LIN {X 0.246,Y -561.732,Z 557.411,A 0.000,B 0.000,C 90.000,E1 109.939} C_DIS
LIN {X 0.060,Y -566.914,Z 557.408,A 0.000,B 0.000,C 90.000,E1 109.450} C_DIS
LIN {X 0.120,Y -571.794,Z 557.405,A 0.000,B 0.000,C 90.000,E1 108.906} C_DIS
LIN {X 0.026,Y -577.234,Z 557.401,A 0.000,B 0.000,C 90.000,E1 108.236} C_DIS
LIN {X 0.253,Y -582.926,Z 557.397,A 0.000,B 0.000,C 90.000,E1 107.402} C_DIS
LIN {X -0.014,Y -588.048,Z 557.392,A 0.000,B 0.000,C 90.000,E1 106.622} C_DIS
LIN {X 0.262,Y -593.519,Z 557.387,A 0.000,B 0.000,C 90.000,E1 105.662} C_DIS
LIN {X -0.063,Y -597.768,Z 557.383,A 0.000,B 0.000,C 90.000,E1 104.898} C_DIS
LIN {X 0.044,Y -603.619,Z 557.376,A 0.000,B 0.000,C 90.000,E1 103.703} C_DIS
LIN {X -0.051,Y -609.222,Z 557.370,A 0.000,B 0.000,C 90.000,E1 102.535} C_DIS
LIN {X -0.030,Y -612.189,Z 557.366,A 0.000,B 0.000,C 90.000,E1 101.883} C_DIS
LIN {X 0.063,Y -616.606,Z 557.360,A 0.000,B 0.000,C 90.000,E1 100.838} C_DIS
LIN {X -0.178,Y -617.680,Z 557.359,A 0.000,B 0.000,C 90.000,E1 100.602} C_DIS
LIN {X 0.226,Y -625.561,Z 557.347,A 0.000,B 0.000,C 90.000,E1 98.511} C_DIS
LIN {X 0.211,Y -630.523,Z 557.340,A 0.000,B 0.000,C 90.000,E1 97.239} C_DIS
LIN {X 0.129,Y -633.410,Z 557.336,A 0.000,B 0.000,C 90.000,E1 96.486} C_DIS
LIN {X -0.264,Y -636.936,Z 557.331,A 0.000,B 0.000,C 90.000,E1 95.511} C_DIS
LIN {X -0.295,Y -639.376,Z 557.326,A 0.000,B 0.000,C 90.000,E1 94.759} C_DIS
LIN {X 0.033,Y -642.183,Z 557.321,A 0.000,B 0.000,C 90.000,E1 93.726} C_DIS
LIN {X -0.005,Y -644.045,Z 557.317,A 0.000,B 0.000,C 90.000,E1 92.980} C_DIS
LIN {X -0.054,Y -645.623,Z 557.312,A 0.000,B 0.000,C 90.000,E1 92.236} C_DIS
LIN {X -0.063,Y -646.957,Z 557.308,A 0.000,B 0.000,C 90.000,E1 91.489} C_DIS
LIN {X 0.141,Y -647.672,Z 557.306,A 0.000,B 0.000,C 90.000,E1 90.974} C_DIS
LIN {X 0.136,Y -648.569,Z 557.301,A 0.000,B 0.000,C 90.000,E1 90.229} C_DIS
LIN {X -0.074,Y -649.177,Z 557.296,A 0.000,B 0.000,C 90.000,E1 89.255} C_DIS
LIN {X -0.289,Y -649.296,Z 557.294,A 0.000,B 0.000,C 90.000,E1 89.026} C_DIS
LIN {X 0.173,Y -649.169,Z 557.289,A 0.000,B 0.000,C 90.000,E1 87.993} C_DIS
LIN {X 0.177,Y -648.851,Z 557.285,A 0.000,B 0.000,C 90.000,E1 87.249} C_DIS
LIN {X -0.014,Y -647.981,Z 557.279,A 0.000,B 0.000,C 90.000,E1 86.274} C_DIS
LIN {X -0.218,Y -646.671,Z 557.274,A 0.000,B 0.000,C 90.000,E1 85.298} C_DIS
LIN {X 0.257,Y -645.100,Z 557.268,A 0.000,B 0.000,C 90.000,E1 84.261} C_DIS
LIN {X 0.246,Y -643.698,Z 557.264,A 0.000,B 0.000,C 90.000,E1 83.514} C_DIS
LIN {X 0.293,Y -641.950,Z 557.260,A 0.000,B 0.000,C 90.000,E1 82.761} C_DIS
LIN {X -0.109,Y -638.605,Z 557.253,A 0.000,B 0.000,C 90.000,E1 81.546} C_DIS
LIN {X -0.104,Y -636.298,Z 557.249,A 0.000,B 0.000,C 90.000,E1 80.792} C_DIS
LIN {X 0.317,Y -633.090,Z 557.243,A 0.000,B 0.000,C 90.000,E1 79.746} C_DIS
LIN {X 0.066,Y -629.496,Z 557.238,A 0.000,B 0.000,C 90.000,E1 78.757} C_DIS
LIN {X 0.095,Y -626.536,Z 557.233,A 0.000,B 0.000,C 90.000,E1 77.993} C_DIS
LIN {X -0.110,Y -622.314,Z 557.228,A 0.000,B 0.000,C 90.000,E1 76.992} C_DIS
LIN {X -0.147,Y -618.764,Z 557.223,A 0.000,B 0.000,C 90.000,E1 76.228} C_DIS
LIN {X 0.042,Y -616.906,Z 557.221,A 0.000,B 0.000,C 90.000,E1 75.825} C_DIS
LIN {X 0.133,Y -613.670,Z 557.218,A 0.000,B 0.000,C 90.000,E1 75.172} C_DIS
LIN {X -0.057,Y -608.690,Z 557.213,A 0.000,B 0.000,C 90.000,E1 74.283} C_DIS
LIN {X -0.085,Y -604.075,Z 557.208,A 0.000,B 0.000,C 90.000,E1 73.504} C_DIS
LIN {X 0.196,Y -600.066,Z 557.205,A 0.000,B 0.000,C 90.000,E1 72.851} C_DIS
LIN {X -0.124,Y -594.698,Z 557.201,A 0.000,B 0.000,C 90.000,E1 72.127} C_DIS
LIN {X -0.047,Y -589.323,Z 557.197,A 0.000,B 0.000,C 90.000,E1 71.456} C_DIS
LIN {X 0.057,Y -584.731,Z 557.194,A 0.000,B 0.000,C 90.000,E1 70.913} C_DIS
LIN {X 0.186,Y -579.750,Z 557.191,A 0.000,B 0.000,C 90.000,E1 70.369} C_DIS
LIN {X -0.324,Y -572.232,Z 557.187,A 0.000,B 0.000,C 90.000,E1 69.699} C_DIS
LIN {X -0.116,Y -568.454,Z 557.185,A 0.000,B 0.000,C 90.000,E1 69.337} C_DIS
LIN {X -0.234,Y -563.003,Z 557.183,A 0.000,B 0.000,C 90.000,E1 68.901} C_DIS
LIN {X -0.053,Y -558.351,Z 557.181,A 0.000,B 0.000,C 90.000,E1 68.539} C_DIS
LIN {X -0.168,Y -553.801,Z 557.179,A 0.000,B 0.000,C 90.000,E1 68.230} C_DIS
LIN {X -0.242,Y -547.427,Z 557.177,A 0.000,B 0.000,C 90.000,E1 67.847} C_DIS
LIN {X -0.026,Y -542.412,Z 557.175,A 0.000,B 0.000,C 90.000,E1 67.539} C_DIS
LIN {X -0.054,Y -537.211,Z 557.174,A 0.000,B 0.000,C 90.000,E1 67.283} C_DIS
LIN {X -0.161,Y -530.311,Z 557.172,A 0.000,B 0.000,C 90.000,E1 66.975} C_DIS
LIN {X 0.245,Y -519.773,Z 557.170,A 0.000,B 0.000,C 90.000,E1 66.485} C_DIS
LIN {X 0.121,Y -505.630,Z 557.167,A 0.000,B 0.000,C 90.000,E1 65.973} C_DIS
LIN {X 0.039,Y -487.939,Z 557.163,A 0.000,B 0.000,C 90.000,E1 65.357} C_DIS
LIN {X 0.281,Y -470.586,Z 557.160,A 0.000,B 0.000,C 90.000,E1 64.717} C_DIS
LIN {X -0.042,Y -459.761,Z 557.157,A 0.000,B 0.000,C 90.000,E1 64.332} C_DIS
LIN {X -0.076,Y -459.738,Z 557.157,A 0.000,B 0.000,C 90.000,E1 64.332} C_DIS
LIN {X -0.044,Y -455.591,Z 557.144,A 0.000,B 0.000,C 90.000,E1 61.975} C_DIS
LIN {X 0.139,Y -452.500,Z 557.137,A 0.000,B 0.000,C 90.000,E1 60.667} C_DIS
LIN {X -0.225,Y -443.899,Z 557.114,A 0.000,B 0.000,C 90.000,E1 56.501} C_DIS
LIN {X 0.022,Y -439.842,Z 557.105,A 0.000,B 0.000,C 90.000,E1 54.848} C_DIS
LIN {X -0.016,Y -439.846,Z 557.105,A 0.000,B 0.000,C 90.000,E1 54.848} C_DIS
LIN {X -0.142,Y -443.210,Z 557.092,A 0.000,B 0.000,C 90.000,E1 52.557} C_DIS
LIN {X 0.164,Y -445.597,Z 557.083,A 0.000,B 0.000,C 90.000,E1 50.884} C_DIS
LIN {X -0.172,Y -447.830,Z 557.074,A 0.000,B 0.000,C 90.000,E1 49.299} C_DIS
LIN {X 0.165,Y -450.382,Z 557.063,A 0.000,B 0.000,C 90.000,E1 47.310} C_DIS
LIN {X -0.114,Y -452.284,Z 557.054,A 0.000,B 0.000,C 90.000,E1 45.729} C_DIS
LIN {X -0.074,Y -453.265,Z 557.049,A 0.000,B 0.000,C 90.000,E1 44.757} C_DIS
LIN {X -0.025,Y -454.053,Z 557.043,A 0.000,B 0.000,C 90.000,E1 43.785} C_DIS
LIN {X -0.261,Y -454.800,Z 557.036,A 0.000,B 0.000,C 90.000,E1 42.528} C_DIS
LIN {X -0.149,Y -455.338,Z 557.029,A 0.000,B 0.000,C 90.000,E1 41.229} C_DIS
LIN {X -0.029,Y -455.588,Z 557.022,A 0.000,B 0.000,C 90.000,E1 39.930} C_DIS
LIN {X 0.152,Y -455.658,Z 557.015,A 0.000,B 0.000,C 90.000,E1 38.624} C_DIS
LIN {X -0.021,Y -455.585,Z 557.008,A 0.000,B 0.000,C 90.000,E1 37.363} C_DIS
LIN {X 0.249,Y -455.272,Z 556.999,A 0.000,B 0.000,C 90.000,E1 35.724} C_DIS
LIN {X 0.246,Y -454.649,Z 556.990,A 0.000,B 0.000,C 90.000,E1 34.119} C_DIS
LIN {X -0.020,Y -454.134,Z 556.981,A 0.000,B 0.000,C 90.000,E1 32.546} C_DIS
LIN {X 0.183,Y -453.549,Z 556.970,A 0.000,B 0.000,C 90.000,E1 30.590} C_DIS
LIN {X 0.040,Y -453.118,Z 556.961,A 0.000,B 0.000,C 90.000,E1 28.999} C_DIS
LIN {X 0.068,Y -452.621,Z 556.952,A 0.000,B 0.000,C 90.000,E1 27.385} C_DIS
LIN {X 0.121,Y -452.373,Z 556.947,A 0.000,B 0.000,C 90.000,E1 26.411} C_DIS
LIN {X 0.115,Y -451.771,Z 556.934,A 0.000,B 0.000,C 90.000,E1 24.155} C_DIS
LIN {X 0.211,Y -451.371,Z 556.924,A 0.000,B 0.000,C 90.000,E1 22.206} C_DIS
LIN {X -0.167,Y -451.125,Z 556.911,A 0.000,B 0.000,C 90.000,E1 19.993} C_DIS
LIN {X 0.141,Y -451.053,Z 556.898,A 0.000,B 0.000,C 90.000,E1 17.692} C_DIS
LIN {X 0.179,Y -451.171,Z 556.886,A 0.000,B 0.000,C 90.000,E1 15.426} C_DIS
LIN {X 0.056,Y -451.742,Z 556.870,A 0.000,B 0.000,C 90.000,E1 12.535} C_DIS
LIN {X -0.002,Y -452.722,Z 556.855,A 0.000,B 0.000,C 90.000,E1 9.962} C_DIS
LIN {X 0.047,Y -453.845,Z 556.843,A 0.000,B 0.000,C 90.000,E1 7.701} C_DIS
LIN {X -0.149,Y -455.117,Z 556.832,A 0.000,B 0.000,C 90.000,E1 5.796} C_DIS
LIN {X -0.007,Y -456.994,Z 556.818,A 0.000,B 0.000,C 90.000,E1 3.212} C_DIS
LIN {X -0.085,Y -460.624,Z 556.797,A 0.000,B 0.000,C 90.000,E1 359.484} C_DIS
LIN {X 0.195,Y -463.699,Z 556.783,A 0.000,B 0.000,C 90.000,E1 356.906} C_DIS
LIN {X 0.192,Y -467.221,Z 556.769,A 0.000,B 0.000,C 90.000,E1 354.375} C_DIS
LIN {X -0.148,Y -469.847,Z 556.758,A 0.000,B 0.000,C 90.000,E1 352.527} C_DIS
LIN {X 0.030,Y -472.470,Z 556.748,A 0.000,B 0.000,C 90.000,E1 350.622} C_DIS
LIN {X 0.086,Y -476.234,Z 556.734,A 0.000,B 0.000,C 90.000,E1 348.117} C_DIS
LIN {X -0.171,Y -479.221,Z 556.724,A 0.000,B 0.000,C 90.000,E1 346.284} C_DIS
LIN {X 0.115,Y -482.419,Z 556.713,A 0.000,B 0.000,C 90.000,E1 344.393} C_DIS
LIN {X 0.000,Y -487.004,Z 556.700,A 0.000,B 0.000,C 90.000,E1 341.945} C_DIS
LIN {X -0.067,Y -490.007,Z 556.691,A 0.000,B 0.000,C 90.000,E1 340.423} C_DIS
LIN {X -0.073,Y -492.971,Z 556.683,A 0.000,B 0.000,C 90.000,E1 338.901} C_DIS
LIN {X 0.150,Y -495.863,Z 556.674,A 0.000,B 0.000,C 90.000,E1 337.358} C_DIS
LIN {X -0.036,Y -498.677,Z 556.666,A 0.000,B 0.000,C 90.000,E1 335.869} C_DIS
LIN {X 0.028,Y -501.386,Z 556.658,A 0.000,B 0.000,C 90.000,E1 334.357} C_DIS
LIN {X -0.087,Y -503.959,Z 556.649,A 0.000,B 0.000,C 90.000,E1 332.871} C_DIS
LIN {X -0.151,Y -506.459,Z 556.641,A 0.000,B 0.000,C 90.000,E1 331.385} C_DIS
LIN {X -0.037,Y -509.523,Z 556.631,A 0.000,B 0.000,C 90.000,E1 329.587} C_DIS
LIN {X 0.152,Y -512.579,Z 556.621,A 0.000,B 0.000,C 90.000,E1 327.788} C_DIS
LIN {X -0.109,Y -515.163,Z 556.613,A 0.000,B 0.000,C 90.000,E1 326.342} C_DIS
LIN {X 0.099,Y -517.782,Z 556.605,A 0.000,B 0.000,C 90.000,E1 324.848} C_DIS
LIN {X -0.253,Y -520.828,Z 556.595,A 0.000,B 0.000,C 90.000,E1 323.130} C_DIS
LIN {X -0.296,Y -525.163,Z 556.582,A 0.000,B 0.000,C 90.000,E1 320.803} C_DIS
LIN {X -0.057,Y -531.883,Z 556.564,A 0.000,B 0.000,C 90.000,E1 317.595} C_DIS
LIN {X -0.283,Y -537.412,Z 556.552,A 0.000,B 0.000,C 90.000,E1 315.324} C_DIS
LIN {X 0.025,Y -540.889,Z 556.544,A 0.000,B 0.000,C 90.000,E1 313.866} C_DIS
LIN {X 0.042,Y -545.394,Z 556.534,A 0.000,B 0.000,C 90.000,E1 312.162} C_DIS
LIN {X 0.055,Y -547.077,Z 556.531,A 0.000,B 0.000,C 90.000,E1 311.595} C_DIS
LIN {X 0.090,Y -547.862,Z 556.530,A 0.000,B 0.000,C 90.000,E1 311.310} C_DIS
LIN {X -0.250,Y -548.890,Z 556.528,A 0.000,B 0.000,C 90.000,E1 311.067} C_DIS
LIN {X -0.208,Y -549.690,Z 556.526,A 0.000,B 0.000,C 90.000,E1 310.782} C_DIS
LIN {X -0.006,Y -550.225,Z 556.526,A 0.000,B 0.000,C 90.000,E1 310.620} C_DIS
LIN {X 0.248,Y -552.243,Z 556.523,A 0.000,B 0.000,C 90.000,E1 310.172} C_DIS
LIN {X -0.031,Y -554.556,Z 556.521,A 0.000,B 0.000,C 90.000,E1 309.850} C_DIS
LIN {X -0.106,Y -557.886,Z 556.519,A 0.000,B 0.000,C 90.000,E1 309.439} C_DIS
LIN {X 0.084,Y -562.492,Z 556.517,A 0.000,B 0.000,C 90.000,E1 308.955} C_DIS
LIN {X 0.103,Y -570.439,Z 556.513,A 0.000,B 0.000,C 90.000,E1 308.302} C_DIS
LIN {X 0.290,Y -580.640,Z 556.509,A 0.000,B 0.000,C 90.000,E1 307.523} C_DIS
LIN {X -0.049,Y -587.620,Z 556.506,A 0.000,B 0.000,C 90.000,E1 306.996} C_DIS
LIN {X -0.167,Y -591.705,Z 556.504,A 0.000,B 0.000,C 90.000,E1 306.664} C_DIS
LIN {X -0.083,Y -596.826,Z 556.501,A 0.000,B 0.000,C 90.000,E1 306.171} C_DIS
LIN {X 0.120,Y -601.796,Z 556.498,A 0.000,B 0.000,C 90.000,E1 305.644} C_DIS
LIN {X -0.162,Y -609.169,Z 556.494,A 0.000,B 0.000,C 90.000,E1 304.898} C_DIS
LIN {X -0.120,Y -615.082,Z 556.490,A 0.000,B 0.000,C 90.000,E1 304.246} C_DIS
LIN {X 0.101,Y -622.014,Z 556.486,A 0.000,B 0.000,C 90.000,E1 303.452} C_DIS
LIN {X -0.118,Y -627.486,Z 556.482,A 0.000,B 0.000,C 90.000,E1 302.832} C_DIS
LIN {X -0.294,Y -632.694,Z 556.479,A 0.000,B 0.000,C 90.000,E1 302.212} C_DIS
LIN {X 0.108,Y -637.456,Z 556.475,A 0.000,B 0.000,C 90.000,E1 301.544} C_DIS
LIN {X 0.008,Y -641.457,Z 556.472,A 0.000,B 0.000,C 90.000,E1 300.924} C_DIS
LIN {X 0.129,Y -644.378,Z 556.469,A 0.000,B 0.000,C 90.000,E1 300.413} C_DIS
LIN {X 0.075,Y -647.411,Z 556.466,A 0.000,B 0.000,C 90.000,E1 299.795} C_DIS
LIN {X -0.238,Y -650.507,Z 556.461,A 0.000,B 0.000,C 90.000,E1 299.077} C_DIS
LIN {X 0.053,Y -653.212,Z 556.457,A 0.000,B 0.000,C 90.000,E1 298.309} C_DIS
LIN {X -0.089,Y -656.682,Z 556.452,A 0.000,B 0.000,C 90.000,E1 297.334} C_DIS
LIN {X 0.029,Y -657.730,Z 556.451,A 0.000,B 0.000,C 90.000,E1 297.078} C_DIS
LIN {X 0.151,Y -658.625,Z 556.449,A 0.000,B 0.000,C 90.000,E1 296.821} C_DIS
LIN {X -0.189,Y -660.124,Z 556.446,A 0.000,B 0.000,C 90.000,E1 296.360} C_DIS
LIN {X -0.059,Y -660.614,Z 556.445,A 0.000,B 0.000,C 90.000,E1 296.104} C_DIS
LIN {X 0.205,Y -660.847,Z 556.442,A 0.000,B 0.000,C 90.000,E1 295.591} C_DIS
LIN {X 0.336,Y -660.497,Z 556.441,A 0.000,B 0.000,C 90.000,E1 295.335} C_DIS
LIN {X 0.402,Y -659.757,Z 556.440,A 0.000,B 0.000,C 90.000,E1 295.207} C_DIS
LIN {X -0.409,Y -659.189,Z 556.440,A 0.000,B 0.000,C 90.000,E1 295.155} C_DIS
LIN {X 0.085,Y -658.729,Z 556.439,A 0.000,B 0.000,C 90.000,E1 294.975} C_DIS
LIN {X 0.213,Y -657.506,Z 556.438,A 0.000,B 0.000,C 90.000,E1 294.719} C_DIS
LIN {X -0.130,Y -653.750,Z 556.435,A 0.000,B 0.000,C 90.000,E1 294.387} C_DIS
LIN {X -0.002,Y -652.702,Z 556.435,A 0.000,B 0.000,C 90.000,E1 294.259} C_DIS
LIN {X 0.050,Y -651.126,Z 556.434,A 0.000,B 0.000,C 90.000,E1 294.131} C_DIS
LIN {X -0.092,Y -644.023,Z 556.432,A 0.000,B 0.000,C 90.000,E1 293.770} C_DIS
LIN {X -0.176,Y -642.024,Z 556.432,A 0.000,B 0.000,C 90.000,E1 293.695} C_DIS
LIN {X -0.331,Y -636.032,Z 556.431,A 0.000,B 0.000,C 90.000,E1 293.515} C_DIS
LIN {X 0.086,Y -632.311,Z 556.430,A 0.000,B 0.000,C 90.000,E1 293.334} C_DIS
LIN {X -0.236,Y -621.253,Z 556.428,A 0.000,B 0.000,C 90.000,E1 293.025} C_DIS
LIN {X 0.165,Y -617.083,Z 556.427,A 0.000,B 0.000,C 90.000,E1 292.845} C_DIS
LIN {X -0.060,Y -587.800,Z 556.422,A 0.000,B 0.000,C 90.000,E1 291.950} C_DIS
LIN {X -0.084,Y -579.731,Z 556.420,A 0.000,B 0.000,C 90.000,E1 291.663} C_DIS
LIN {X -0.040,Y -574.163,Z 556.419,A 0.000,B 0.000,C 90.000,E1 291.408} C_DIS
LIN {X -0.185,Y -569.857,Z 556.417,A 0.000,B 0.000,C 90.000,E1 291.153} C_DIS
LIN {X 0.029,Y -568.280,Z 556.416,A 0.000,B 0.000,C 90.000,E1 290.918} C_DIS
LIN {X 0.013,Y -567.693,Z 556.415,A 0.000,B 0.000,C 90.000,E1 290.663} C_DIS
LIN {X -0.039,Y -567.413,Z 556.412,A 0.000,B 0.000,C 90.000,E1 290.120} C_DIS
LIN {X 0.198,Y -567.328,Z 556.404,A 0.000,B 0.000,C 90.000,E1 288.725} C_DIS
LIN {X 0.097,Y -567.175,Z 556.398,A 0.000,B 0.000,C 90.000,E1 287.638} C_DIS
LIN {X 0.151,Y -566.751,Z 556.390,A 0.000,B 0.000,C 90.000,E1 286.260} C_DIS
LIN {X -0.193,Y -565.873,Z 556.381,A 0.000,B 0.000,C 90.000,E1 284.647} C_DIS
LIN {X 0.094,Y -565.058,Z 556.374,A 0.000,B 0.000,C 90.000,E1 283.244} C_DIS
LIN {X -0.053,Y -564.308,Z 556.366,A 0.000,B 0.000,C 90.000,E1 281.883} C_DIS
LIN {X 0.106,Y -563.565,Z 556.358,A 0.000,B 0.000,C 90.000,E1 280.489} C_DIS
LIN {X 0.020,Y -562.571,Z 556.348,A 0.000,B 0.000,C 90.000,E1 278.568} C_DIS
LIN {X -0.256,Y -561.703,Z 556.337,A 0.000,B 0.000,C 90.000,E1 276.663} C_DIS
LIN {X 0.114,Y -561.352,Z 556.332,A 0.000,B 0.000,C 90.000,E1 275.796} C_DIS
LIN {X 0.088,Y -560.796,Z 556.325,A 0.000,B 0.000,C 90.000,E1 274.416} C_DIS
LIN {X 0.047,Y -560.239,Z 556.317,A 0.000,B 0.000,C 90.000,E1 273.037} C_DIS
LIN {X 0.142,Y -559.423,Z 556.306,A 0.000,B 0.000,C 90.000,E1 271.088} C_DIS
LIN {X 0.034,Y -558.715,Z 556.298,A 0.000,B 0.000,C 90.000,E1 269.714} C_DIS
LIN {X 0.096,Y -557.677,Z 556.288,A 0.000,B 0.000,C 90.000,E1 267.764} C_DIS
LIN {X -0.029,Y -556.879,Z 556.280,A 0.000,B 0.000,C 90.000,E1 266.388} C_DIS
LIN {X -0.066,Y -555.872,Z 556.271,A 0.000,B 0.000,C 90.000,E1 264.723} C_DIS
LIN {X -0.079,Y -554.755,Z 556.261,A 0.000,B 0.000,C 90.000,E1 263.053} C_DIS
LIN {X -0.092,Y -553.759,Z 556.254,A 0.000,B 0.000,C 90.000,E1 261.659} C_DIS
LIN {X -0.204,Y -552.293,Z 556.246,A 0.000,B 0.000,C 90.000,E1 260.274} C_DIS
LIN {X 0.180,Y -549.638,Z 556.233,A 0.000,B 0.000,C 90.000,E1 257.993} C_DIS
LIN {X -0.252,Y -547.788,Z 556.224,A 0.000,B 0.000,C 90.000,E1 256.353} C_DIS
LIN {X 0.068,Y -545.677,Z 556.215,A 0.000,B 0.000,C 90.000,E1 254.629} C_DIS
LIN {X -0.049,Y -544.507,Z 556.210,A 0.000,B 0.000,C 90.000,E1 253.795} C_DIS
LIN {X -0.327,Y -541.934,Z 556.201,A 0.000,B 0.000,C 90.000,E1 252.127} C_DIS
LIN {X -0.094,Y -540.044,Z 556.194,A 0.000,B 0.000,C 90.000,E1 250.967} C_DIS
LIN {X -0.066,Y -538.087,Z 556.188,A 0.000,B 0.000,C 90.000,E1 249.826} C_DIS
LIN {X -0.178,Y -535.280,Z 556.180,A 0.000,B 0.000,C 90.000,E1 248.411} C_DIS
LIN {X 0.154,Y -532.886,Z 556.174,A 0.000,B 0.000,C 90.000,E1 247.230} C_DIS
LIN {X -0.035,Y -530.386,Z 556.167,A 0.000,B 0.000,C 90.000,E1 246.102} C_DIS
LIN {X -0.259,Y -527.720,Z 556.161,A 0.000,B 0.000,C 90.000,E1 244.973} C_DIS
LIN {X -0.133,Y -524.130,Z 556.153,A 0.000,B 0.000,C 90.000,E1 243.512} C_DIS
LIN {X 0.159,Y -520.389,Z 556.145,A 0.000,B 0.000,C 90.000,E1 242.025} C_DIS
LIN {X -0.077,Y -516.643,Z 556.137,A 0.000,B 0.000,C 90.000,E1 240.589} C_DIS
LIN {X -0.037,Y -513.407,Z 556.130,A 0.000,B 0.000,C 90.000,E1 239.410} C_DIS
LIN {X -0.252,Y -507.950,Z 556.120,A 0.000,B 0.000,C 90.000,E1 237.661} C_DIS
LIN {X -0.127,Y -501.004,Z 556.107,A 0.000,B 0.000,C 90.000,E1 235.261} C_DIS
LIN {X -0.187,Y -493.404,Z 556.092,A 0.000,B 0.000,C 90.000,E1 232.557} C_DIS
LIN {X 0.064,Y -489.298,Z 556.083,A 0.000,B 0.000,C 90.000,E1 231.009} C_DIS
LIN {X 0.236,Y -485.378,Z 556.075,A 0.000,B 0.000,C 90.000,E1 229.461} C_DIS
LIN {X 0.081,Y -480.635,Z 556.065,A 0.000,B 0.000,C 90.000,E1 227.634} C_DIS
LIN {X 0.013,Y -474.464,Z 556.051,A 0.000,B 0.000,C 90.000,E1 225.162} C_DIS
LIN {X -0.167,Y -470.788,Z 556.042,A 0.000,B 0.000,C 90.000,E1 223.623} C_DIS
LIN {X 0.091,Y -465.675,Z 556.030,A 0.000,B 0.000,C 90.000,E1 221.391} C_DIS
LIN {X -0.093,Y -460.693,Z 556.018,A 0.000,B 0.000,C 90.000,E1 219.197} C_DIS
LIN {X -0.083,Y -456.527,Z 556.007,A 0.000,B 0.000,C 90.000,E1 217.282} C_DIS
LIN {X 0.082,Y -451.106,Z 555.993,A 0.000,B 0.000,C 90.000,E1 214.692} C_DIS
LIN {X 0.137,Y -446.542,Z 555.980,A 0.000,B 0.000,C 90.000,E1 212.418} C_DIS
LIN {X 0.251,Y -441.609,Z 555.966,A 0.000,B 0.000,C 90.000,E1 209.795} C_DIS
LIN {X -0.056,Y -436.924,Z 555.951,A 0.000,B 0.000,C 90.000,E1 207.206} C_DIS
LIN {X 0.224,Y -434.723,Z 555.944,A 0.000,B 0.000,C 90.000,E1 205.848} C_DIS
LIN {X 0.092,Y -431.993,Z 555.935,A 0.000,B 0.000,C 90.000,E1 204.207} C_DIS
LIN {X -0.086,Y -428.371,Z 555.922,A 0.000,B 0.000,C 90.000,E1 201.897} C_DIS
LIN {X -0.083,Y -424.536,Z 555.907,A 0.000,B 0.000,C 90.000,E1 199.214} C_DIS
LIN {X 0.052,Y -422.347,Z 555.897,A 0.000,B 0.000,C 90.000,E1 197.511} C_DIS
LIN {X 0.055,Y -419.752,Z 555.886,A 0.000,B 0.000,C 90.000,E1 195.481} C_DIS
LIN {X 0.138,Y -417.820,Z 555.877,A 0.000,B 0.000,C 90.000,E1 193.772} C_DIS
LIN {X -0.009,Y -416.441,Z 555.871,A 0.000,B 0.000,C 90.000,E1 192.771} C_DIS
LIN {X -0.165,Y -411.538,Z 555.850,A 0.000,B 0.000,C 90.000,E1 189.029} C_DIS
LIN {X -0.031,Y -408.211,Z 555.833,A 0.000,B 0.000,C 90.000,E1 185.910} C_DIS
LIN {X -0.056,Y -406.914,Z 555.825,A 0.000,B 0.000,C 90.000,E1 184.531} C_DIS
LIN {X 0.142,Y -403.757,Z 555.806,A 0.000,B 0.000,C 90.000,E1 181.031} C_DIS
LIN {X -0.160,Y -401.745,Z 555.788,A 0.000,B 0.000,C 90.000,E1 177.936} C_DIS
LIN {X -0.043,Y -400.547,Z 555.773,A 0.000,B 0.000,C 90.000,E1 175.122} C_DIS
LIN {X 0.088,Y -399.857,Z 555.755,A 0.000,B 0.000,C 90.000,E1 171.951} C_DIS
LIN {X 0.009,Y -399.774,Z 555.744,A 0.000,B 0.000,C 90.000,E1 169.859} C_DIS
LIN {X -0.035,Y -399.964,Z 555.728,A 0.000,B 0.000,C 90.000,E1 167.061} C_DIS
LIN {X 0.127,Y -400.385,Z 555.716,A 0.000,B 0.000,C 90.000,E1 164.936} C_DIS
LIN {X -0.193,Y -401.346,Z 555.701,A 0.000,B 0.000,C 90.000,E1 162.181} C_DIS
LIN {X 0.059,Y -402.428,Z 555.687,A 0.000,B 0.000,C 90.000,E1 159.699} C_DIS
LIN {X -0.124,Y -403.678,Z 555.674,A 0.000,B 0.000,C 90.000,E1 157.283} C_DIS
LIN {X -0.111,Y -405.118,Z 555.660,A 0.000,B 0.000,C 90.000,E1 154.845} C_DIS
LIN {X 0.014,Y -406.362,Z 555.649,A 0.000,B 0.000,C 90.000,E1 152.743} C_DIS
LIN {X 0.077,Y -407.396,Z 555.639,A 0.000,B 0.000,C 90.000,E1 151.001} C_DIS
LIN {X -0.003,Y -408.278,Z 555.629,A 0.000,B 0.000,C 90.000,E1 149.282} C_DIS
LIN {X -0.119,Y -408.845,Z 555.622,A 0.000,B 0.000,C 90.000,E1 147.916} C_DIS
LIN {X 0.122,Y -409.336,Z 555.614,A 0.000,B 0.000,C 90.000,E1 146.501} C_DIS
LIN {X 0.021,Y -409.833,Z 555.606,A 0.000,B 0.000,C 90.000,E1 145.135} C_DIS
LIN {X 0.137,Y -410.260,Z 555.595,A 0.000,B 0.000,C 90.000,E1 143.050} C_DIS
LIN {X 0.108,Y -410.492,Z 555.585,A 0.000,B 0.000,C 90.000,E1 141.331} C_DIS
LIN {X 0.013,Y -410.605,Z 555.576,A 0.000,B 0.000,C 90.000,E1 139.622} C_DIS
LIN {X 0.037,Y -410.644,Z 555.564,A 0.000,B 0.000,C 90.000,E1 137.553} C_DIS
LIN {X 0.042,Y -410.739,Z 555.553,A 0.000,B 0.000,C 90.000,E1 135.486} C_DIS
LIN {X -0.099,Y -410.948,Z 555.543,A 0.000,B 0.000,C 90.000,E1 133.785} C_DIS
LIN {X 0.054,Y -411.122,Z 555.534,A 0.000,B 0.000,C 90.000,E1 132.043} C_DIS
LIN {X -0.194,Y -411.095,Z 555.526,A 0.000,B 0.000,C 90.000,E1 130.701} C_DIS
LIN {X 0.143,Y -410.907,Z 555.518,A 0.000,B 0.000,C 90.000,E1 129.277} C_DIS
LIN {X 0.055,Y -410.617,Z 555.513,A 0.000,B 0.000,C 90.000,E1 128.257} C_DIS
LIN {X -0.211,Y -410.410,Z 555.510,A 0.000,B 0.000,C 90.000,E1 127.729} C_DIS
LIN {X 0.075,Y -410.416,Z 555.509,A 0.000,B 0.000,C 90.000,E1 127.684} C_DIS
LIN {X -0.190,Y -415.820,Z 555.499,A 0.000,B 0.000,C 90.000,E1 125.884} C_DIS
LIN {X -0.086,Y -425.279,Z 555.479,A 0.000,B 0.000,C 90.000,E1 122.133} C_DIS
LIN {X -0.152,Y -430.286,Z 555.469,A 0.000,B 0.000,C 90.000,E1 120.463} C_DIS
LIN {X -0.154,Y -431.177,Z 555.467,A 0.000,B 0.000,C 90.000,E1 120.129} C_DIS
LIN {X -0.135,Y -440.845,Z 555.446,A 0.000,B 0.000,C 90.000,E1 116.283} C_DIS
LIN {X 0.221,Y -440.859,Z 555.446,A 0.000,B 0.000,C 90.000,E1 116.232} C_DIS
LIN {X 0.181,Y -440.903,Z 555.446,A 0.000,B 0.000,C 90.000,E1 116.232} C_DIS
LIN {X -0.201,Y -466.035,Z 555.440,A 0.000,B 0.000,C 90.000,E1 115.155} C_DIS
LIN {X -0.089,Y -481.629,Z 555.436,A 0.000,B 0.000,C 90.000,E1 114.463} C_DIS
LIN {X 0.121,Y -495.089,Z 555.432,A 0.000,B 0.000,C 90.000,E1 113.823} C_DIS
LIN {X 0.140,Y -505.135,Z 555.430,A 0.000,B 0.000,C 90.000,E1 113.334} C_DIS
LIN {X -0.211,Y -516.700,Z 555.426,A 0.000,B 0.000,C 90.000,E1 112.770} C_DIS
LIN {X 0.174,Y -521.670,Z 555.425,A 0.000,B 0.000,C 90.000,E1 112.461} C_DIS
LIN {X -0.010,Y -532.926,Z 555.421,A 0.000,B 0.000,C 90.000,E1 111.844} C_DIS
LIN {X 0.006,Y -539.270,Z 555.419,A 0.000,B 0.000,C 90.000,E1 111.461} C_DIS
LIN {X 0.146,Y -545.378,Z 555.417,A 0.000,B 0.000,C 90.000,E1 111.046} C_DIS
LIN {X 0.291,Y -551.315,Z 555.415,A 0.000,B 0.000,C 90.000,E1 110.610} C_DIS
LIN {X 0.091,Y -555.703,Z 555.413,A 0.000,B 0.000,C 90.000,E1 110.301} C_DIS
LIN {X -0.189,Y -561.189,Z 555.410,A 0.000,B 0.000,C 90.000,E1 109.866} C_DIS
LIN {X 0.259,Y -566.391,Z 555.408,A 0.000,B 0.000,C 90.000,E1 109.322} C_DIS
LIN {X -0.078,Y -571.276,Z 555.405,A 0.000,B 0.000,C 90.000,E1 108.833} C_DIS
LIN {X 0.330,Y -577.300,Z 555.401,A 0.000,B 0.000,C 90.000,E1 108.055} C_DIS
LIN {X -0.118,Y -580.266,Z 555.398,A 0.000,B 0.000,C 90.000,E1 107.692} C_DIS
LIN {X 0.087,Y -582.263,Z 555.397,A 0.000,B 0.000,C 90.000,E1 107.402} C_DIS
LIN {X -0.268,Y -588.417,Z 555.392,A 0.000,B 0.000,C 90.000,E1 106.496} C_DIS
LIN {X -0.153,Y -594.014,Z 555.386,A 0.000,B 0.000,C 90.000,E1 105.552} C_DIS
LIN {X 0.191,Y -598.977,Z 555.381,A 0.000,B 0.000,C 90.000,E1 104.592} C_DIS
LIN {X -0.145,Y -603.623,Z 555.376,A 0.000,B 0.000,C 90.000,E1 103.703} C_DIS
LIN {X -0.240,Y -609.386,Z 555.370,A 0.000,B 0.000,C 90.000,E1 102.535} C_DIS
LIN {X 0.195,Y -612.997,Z 555.365,A 0.000,B 0.000,C 90.000,E1 101.715} C_DIS
LIN {X 0.057,Y -616.393,Z 555.361,A 0.000,B 0.000,C 90.000,E1 100.950} C_DIS
LIN {X 0.071,Y -618.507,Z 555.358,A 0.000,B 0.000,C 90.000,E1 100.433} C_DIS
LIN {X 0.295,Y -627.505,Z 555.345,A 0.000,B 0.000,C 90.000,E1 98.106} C_DIS
LIN {X 0.313,Y -632.469,Z 555.338,A 0.000,B 0.000,C 90.000,E1 96.834} C_DIS
LIN {X -0.025,Y -636.225,Z 555.333,A 0.000,B 0.000,C 90.000,E1 95.853} C_DIS
LIN {X 0.261,Y -639.538,Z 555.327,A 0.000,B 0.000,C 90.000,E1 94.821} C_DIS
LIN {X -0.189,Y -641.071,Z 555.324,A 0.000,B 0.000,C 90.000,E1 94.359} C_DIS
LIN {X -0.234,Y -643.150,Z 555.320,A 0.000,B 0.000,C 90.000,E1 93.612} C_DIS
LIN {X -0.263,Y -644.999,Z 555.316,A 0.000,B 0.000,C 90.000,E1 92.865} C_DIS
LIN {X 0.121,Y -647.041,Z 555.310,A 0.000,B 0.000,C 90.000,E1 91.835} C_DIS
LIN {X 0.125,Y -648.219,Z 555.306,A 0.000,B 0.000,C 90.000,E1 91.088} C_DIS
LIN {X -0.090,Y -649.363,Z 555.301,A 0.000,B 0.000,C 90.000,E1 90.115} C_DIS
LIN {X -0.079,Y -649.780,Z 555.297,A 0.000,B 0.000,C 90.000,E1 89.370} C_DIS
LIN {X 0.148,Y -649.957,Z 555.294,A 0.000,B 0.000,C 90.000,E1 88.854} C_DIS
LIN {X -0.031,Y -649.797,Z 555.288,A 0.000,B 0.000,C 90.000,E1 87.879} C_DIS
LIN {X -0.022,Y -649.358,Z 555.284,A 0.000,B 0.000,C 90.000,E1 87.135} C_DIS
LIN {X -0.208,Y -648.422,Z 555.279,A 0.000,B 0.000,C 90.000,E1 86.159} C_DIS
LIN {X 0.291,Y -647.050,Z 555.273,A 0.000,B 0.000,C 90.000,E1 85.122} C_DIS
LIN {X 0.306,Y -645.818,Z 555.269,A 0.000,B 0.000,C 90.000,E1 84.375} C_DIS
LIN {X -0.098,Y -644.939,Z 555.266,A 0.000,B 0.000,C 90.000,E1 83.913} C_DIS
LIN {X 0.136,Y -643.893,Z 555.263,A 0.000,B 0.000,C 90.000,E1 83.394} C_DIS
LIN {X -0.061,Y -641.344,Z 555.258,A 0.000,B 0.000,C 90.000,E1 82.413} C_DIS
LIN {X -0.028,Y -639.310,Z 555.254,A 0.000,B 0.000,C 90.000,E1 81.659} C_DIS
LIN {X -0.292,Y -636.183,Z 555.248,A 0.000,B 0.000,C 90.000,E1 80.679} C_DIS
LIN {X -0.205,Y -633.727,Z 555.244,A 0.000,B 0.000,C 90.000,E1 79.916} C_DIS
LIN {X 0.181,Y -630.109,Z 555.238,A 0.000,B 0.000,C 90.000,E1 78.870} C_DIS
LIN {X -0.328,Y -628.146,Z 555.235,A 0.000,B 0.000,C 90.000,E1 78.409} C_DIS
LIN {X 0.093,Y -623.900,Z 555.230,A 0.000,B 0.000,C 90.000,E1 77.353} C_DIS
LIN {X 0.030,Y -619.853,Z 555.225,A 0.000,B 0.000,C 90.000,E1 76.464} C_DIS
LIN {X -0.001,Y -616.710,Z 555.221,A 0.000,B 0.000,C 90.000,E1 75.825} C_DIS
LIN {X 0.086,Y -613.352,Z 555.218,A 0.000,B 0.000,C 90.000,E1 75.172} C_DIS
LIN {X 0.102,Y -609.003,Z 555.213,A 0.000,B 0.000,C 90.000,E1 74.393} C_DIS
LIN {X 0.078,Y -604.301,Z 555.209,A 0.000,B 0.000,C 90.000,E1 73.614} C_DIS
LIN {X 0.126,Y -599.244,Z 555.205,A 0.000,B 0.000,C 90.000,E1 72.851} C_DIS
LIN {X -0.214,Y -596.277,Z 555.203,A 0.000,B 0.000,C 90.000,E1 72.489} C_DIS
LIN {X 0.239,Y -594.386,Z 555.201,A 0.000,B 0.000,C 90.000,E1 72.181} C_DIS
LIN {X -0.142,Y -589.088,Z 555.198,A 0.000,B 0.000,C 90.000,E1 71.583} C_DIS
LIN {X -0.055,Y -583.677,Z 555.194,A 0.000,B 0.000,C 90.000,E1 70.967} C_DIS
LIN {X 0.146,Y -579.925,Z 555.192,A 0.000,B 0.000,C 90.000,E1 70.550} C_DIS
LIN {X -0.080,Y -573.237,Z 555.189,A 0.000,B 0.000,C 90.000,E1 69.934} C_DIS
LIN {X -0.178,Y -569.149,Z 555.186,A 0.000,B 0.000,C 90.000,E1 69.571} C_DIS
LIN {X -0.016,Y -563.303,Z 555.184,A 0.000,B 0.000,C 90.000,E1 69.082} C_DIS
LIN {X -0.084,Y -557.125,Z 555.181,A 0.000,B 0.000,C 90.000,E1 68.646} C_DIS
LIN {X -0.161,Y -552.412,Z 555.180,A 0.000,B 0.000,C 90.000,E1 68.337} C_DIS
LIN {X 0.048,Y -545.655,Z 555.177,A 0.000,B 0.000,C 90.000,E1 67.922} C_DIS
LIN {X -0.123,Y -540.706,Z 555.176,A 0.000,B 0.000,C 90.000,E1 67.667} C_DIS
LIN {X 0.178,Y -533.644,Z 555.174,A 0.000,B 0.000,C 90.000,E1 67.305} C_DIS
LIN {X -0.268,Y -526.607,Z 555.172,A 0.000,B 0.000,C 90.000,E1 67.050} C_DIS
LIN {X -0.014,Y -517.922,Z 555.170,A 0.000,B 0.000,C 90.000,E1 66.666} C_DIS
LIN {X -0.297,Y -503.467,Z 555.168,A 0.000,B 0.000,C 90.000,E1 66.177} C_DIS
LIN {X -0.073,Y -489.197,Z 555.165,A 0.000,B 0.000,C 90.000,E1 65.665} C_DIS
LIN {X 0.055,Y -471.887,Z 555.161,A 0.000,B 0.000,C 90.000,E1 65.049} C_DIS
LIN {X 0.178,Y -460.361,Z 555.159,A 0.000,B 0.000,C 90.000,E1 64.588} C_DIS
LIN {X 0.143,Y -460.296,Z 555.159,A 0.000,B 0.000,C 90.000,E1 64.588} C_DIS
LIN {X -0.076,Y -455.585,Z 555.144,A 0.000,B 0.000,C 90.000,E1 61.975} C_DIS
LIN {X 0.108,Y -452.491,Z 555.137,A 0.000,B 0.000,C 90.000,E1 60.667} C_DIS
LIN {X -0.257,Y -443.890,Z 555.114,A 0.000,B 0.000,C 90.000,E1 56.501} C_DIS
LIN {X -0.083,Y -440.225,Z 555.106,A 0.000,B 0.000,C 90.000,E1 55.022} C_DIS
LIN {X -0.122,Y -440.217,Z 555.106,A 0.000,B 0.000,C 90.000,E1 55.022} C_DIS
LIN {X 0.158,Y -443.438,Z 555.094,A 0.000,B 0.000,C 90.000,E1 52.844} C_DIS
LIN {X -0.155,Y -445.922,Z 555.085,A 0.000,B 0.000,C 90.000,E1 51.251} C_DIS
LIN {X -0.145,Y -448.193,Z 555.076,A 0.000,B 0.000,C 90.000,E1 49.622} C_DIS
LIN {X -0.136,Y -449.935,Z 555.068,A 0.000,B 0.000,C 90.000,E1 48.324} C_DIS
LIN {X -0.102,Y -451.669,Z 555.061,A 0.000,B 0.000,C 90.000,E1 47.025} C_DIS
LIN {X -0.061,Y -453.173,Z 555.054,A 0.000,B 0.000,C 90.000,E1 45.729} C_DIS
LIN {X 0.008,Y -454.356,Z 555.047,A 0.000,B 0.000,C 90.000,E1 44.433} C_DIS
LIN {X 0.049,Y -454.899,Z 555.043,A 0.000,B 0.000,C 90.000,E1 43.785} C_DIS
LIN {X -0.175,Y -455.598,Z 555.036,A 0.000,B 0.000,C 90.000,E1 42.528} C_DIS
LIN {X -0.049,Y -456.117,Z 555.029,A 0.000,B 0.000,C 90.000,E1 41.229} C_DIS
LIN {X 0.082,Y -456.369,Z 555.022,A 0.000,B 0.000,C 90.000,E1 39.930} C_DIS
LIN {X -0.081,Y -456.390,Z 555.015,A 0.000,B 0.000,C 90.000,E1 38.669} C_DIS
LIN {X -0.158,Y -456.222,Z 555.006,A 0.000,B 0.000,C 90.000,E1 37.076} C_DIS
LIN {X -0.239,Y -455.956,Z 554.999,A 0.000,B 0.000,C 90.000,E1 35.804} C_DIS
LIN {X 0.131,Y -455.205,Z 554.988,A 0.000,B 0.000,C 90.000,E1 33.833} C_DIS
LIN {X -0.129,Y -454.658,Z 554.979,A 0.000,B 0.000,C 90.000,E1 32.260} C_DIS
LIN {X -0.151,Y -454.063,Z 554.968,A 0.000,B 0.000,C 90.000,E1 30.335} C_DIS
LIN {X 0.117,Y -453.598,Z 554.960,A 0.000,B 0.000,C 90.000,E1 28.693} C_DIS
LIN {X -0.154,Y -453.006,Z 554.949,A 0.000,B 0.000,C 90.000,E1 26.796} C_DIS
LIN {X 0.043,Y -452.304,Z 554.936,A 0.000,B 0.000,C 90.000,E1 24.515} C_DIS
LIN {X -0.028,Y -451.894,Z 554.926,A 0.000,B 0.000,C 90.000,E1 22.589} C_DIS
LIN {X -0.111,Y -451.581,Z 554.915,A 0.000,B 0.000,C 90.000,E1 20.663} C_DIS
LIN {X 0.211,Y -451.401,Z 554.902,A 0.000,B 0.000,C 90.000,E1 18.362} C_DIS
LIN {X 0.142,Y -451.484,Z 554.888,A 0.000,B 0.000,C 90.000,E1 15.788} C_DIS
LIN {X -0.104,Y -451.992,Z 554.870,A 0.000,B 0.000,C 90.000,E1 12.591} C_DIS
LIN {X 0.081,Y -452.806,Z 554.857,A 0.000,B 0.000,C 90.000,E1 10.310} C_DIS
LIN {X -0.106,Y -454.050,Z 554.843,A 0.000,B 0.000,C 90.000,E1 7.757} C_DIS
LIN {X -0.134,Y -455.496,Z 554.831,A 0.000,B 0.000,C 90.000,E1 5.511} C_DIS
LIN {X 0.053,Y -457.374,Z 554.816,A 0.000,B 0.000,C 90.000,E1 2.922} C_DIS
LIN {X 0.118,Y -461.114,Z 554.795,A 0.000,B 0.000,C 90.000,E1 359.141} C_DIS
LIN {X 0.186,Y -464.638,Z 554.779,A 0.000,B 0.000,C 90.000,E1 356.274} C_DIS
LIN {X 0.199,Y -467.315,Z 554.769,A 0.000,B 0.000,C 90.000,E1 354.375} C_DIS
LIN {X -0.138,Y -469.909,Z 554.758,A 0.000,B 0.000,C 90.000,E1 352.527} C_DIS
LIN {X -0.133,Y -472.966,Z 554.746,A 0.000,B 0.000,C 90.000,E1 350.330} C_DIS
LIN {X 0.098,Y -476.273,Z 554.734,A 0.000,B 0.000,C 90.000,E1 348.117} C_DIS
LIN {X -0.158,Y -479.285,Z 554.724,A 0.000,B 0.000,C 90.000,E1 346.284} C_DIS
LIN {X -0.016,Y -483.016,Z 554.712,A 0.000,B 0.000,C 90.000,E1 344.102} C_DIS
LIN {X 0.016,Y -487.071,Z 554.700,A 0.000,B 0.000,C 90.000,E1 341.945} C_DIS
LIN {X -0.049,Y -490.072,Z 554.691,A 0.000,B 0.000,C 90.000,E1 340.423} C_DIS
LIN {X -0.014,Y -493.635,Z 554.681,A 0.000,B 0.000,C 90.000,E1 338.592} C_DIS
LIN {X 0.222,Y -496.505,Z 554.673,A 0.000,B 0.000,C 90.000,E1 337.050} C_DIS
LIN {X 0.252,Y -499.299,Z 554.664,A 0.000,B 0.000,C 90.000,E1 335.537} C_DIS
LIN {X -0.115,Y -502.003,Z 554.656,A 0.000,B 0.000,C 90.000,E1 334.076} C_DIS
LIN {X 0.008,Y -504.586,Z 554.648,A 0.000,B 0.000,C 90.000,E1 332.564} C_DIS
LIN {X -0.176,Y -507.620,Z 554.638,A 0.000,B 0.000,C 90.000,E1 330.795} C_DIS
LIN {X -0.036,Y -510.684,Z 554.628,A 0.000,B 0.000,C 90.000,E1 328.997} C_DIS
LIN {X -0.175,Y -513.250,Z 554.620,A 0.000,B 0.000,C 90.000,E1 327.533} C_DIS
LIN {X 0.284,Y -515.856,Z 554.611,A 0.000,B 0.000,C 90.000,E1 326.008} C_DIS
LIN {X 0.078,Y -518.496,Z 554.603,A 0.000,B 0.000,C 90.000,E1 324.562} C_DIS
LIN {X -0.258,Y -521.544,Z 554.593,A 0.000,B 0.000,C 90.000,E1 322.844} C_DIS
LIN {X -0.243,Y -525.370,Z 554.582,A 0.000,B 0.000,C 90.000,E1 320.803} C_DIS
LIN {X 0.004,Y -532.076,Z 554.564,A 0.000,B 0.000,C 90.000,E1 317.595} C_DIS
LIN {X -0.216,Y -537.555,Z 554.552,A 0.000,B 0.000,C 90.000,E1 315.324} C_DIS
LIN {X -0.277,Y -540.366,Z 554.545,A 0.000,B 0.000,C 90.000,E1 314.190} C_DIS
LIN {X 0.132,Y -547.041,Z 554.531,A 0.000,B 0.000,C 90.000,E1 311.595} C_DIS
LIN {X 0.034,Y -549.807,Z 554.526,A 0.000,B 0.000,C 90.000,E1 310.620} C_DIS
LIN {X 0.235,Y -550.464,Z 554.525,A 0.000,B 0.000,C 90.000,E1 310.458} C_DIS
LIN {X -0.286,Y -551.901,Z 554.523,A 0.000,B 0.000,C 90.000,E1 310.092} C_DIS
LIN {X -0.229,Y -553.644,Z 554.521,A 0.000,B 0.000,C 90.000,E1 309.806} C_DIS
LIN {X 0.084,Y -554.571,Z 554.520,A 0.000,B 0.000,C 90.000,E1 309.564} C_DIS
LIN {X 0.120,Y -558.306,Z 554.517,A 0.000,B 0.000,C 90.000,E1 309.072} C_DIS
LIN {X 0.247,Y -561.227,Z 554.515,A 0.000,B 0.000,C 90.000,E1 308.749} C_DIS
LIN {X 0.096,Y -565.326,Z 554.513,A 0.000,B 0.000,C 90.000,E1 308.382} C_DIS
LIN {X 0.026,Y -569.837,Z 554.511,A 0.000,B 0.000,C 90.000,E1 308.016} C_DIS
LIN {X 0.285,Y -579.728,Z 554.507,A 0.000,B 0.000,C 90.000,E1 307.237} C_DIS
LIN {X -0.126,Y -586.712,Z 554.504,A 0.000,B 0.000,C 90.000,E1 306.710} C_DIS
LIN {X 0.071,Y -589.450,Z 554.503,A 0.000,B 0.000,C 90.000,E1 306.457} C_DIS
LIN {X 0.122,Y -594.661,Z 554.500,A 0.000,B 0.000,C 90.000,E1 305.964} C_DIS
LIN {X 0.026,Y -599.638,Z 554.497,A 0.000,B 0.000,C 90.000,E1 305.471} C_DIS
LIN {X 0.025,Y -608.135,Z 554.492,A 0.000,B 0.000,C 90.000,E1 304.565} C_DIS
LIN {X 0.317,Y -617.599,Z 554.486,A 0.000,B 0.000,C 90.000,E1 303.499} C_DIS
LIN {X 0.143,Y -624.274,Z 554.482,A 0.000,B 0.000,C 90.000,E1 302.752} C_DIS
LIN {X -0.049,Y -631.699,Z 554.477,A 0.000,B 0.000,C 90.000,E1 301.878} C_DIS
LIN {X -0.213,Y -635.573,Z 554.474,A 0.000,B 0.000,C 90.000,E1 301.386} C_DIS
LIN {X 0.212,Y -639.669,Z 554.471,A 0.000,B 0.000,C 90.000,E1 300.718} C_DIS
LIN {X -0.234,Y -642.660,Z 554.468,A 0.000,B 0.000,C 90.000,E1 300.256} C_DIS
LIN {X -0.028,Y -646.279,Z 554.464,A 0.000,B 0.000,C 90.000,E1 299.489} C_DIS
LIN {X -0.035,Y -649.223,Z 554.460,A 0.000,B 0.000,C 90.000,E1 298.743} C_DIS
LIN {X 0.193,Y -656.347,Z 554.449,A 0.000,B 0.000,C 90.000,E1 296.744} C_DIS
LIN {X 0.309,Y -657.168,Z 554.447,A 0.000,B 0.000,C 90.000,E1 296.488} C_DIS
LIN {X -0.163,Y -657.758,Z 554.446,A 0.000,B 0.000,C 90.000,E1 296.283} C_DIS
LIN {X -0.207,Y -658.290,Z 554.443,A 0.000,B 0.000,C 90.000,E1 295.796} C_DIS
LIN {X -0.082,Y -658.318,Z 554.442,A 0.000,B 0.000,C 90.000,E1 295.540} C_DIS
LIN {X 0.167,Y -656.837,Z 554.439,A 0.000,B 0.000,C 90.000,E1 295.027} C_DIS
LIN {X 0.228,Y -656.372,Z 554.438,A 0.000,B 0.000,C 90.000,E1 294.899} C_DIS
LIN {X 0.288,Y -655.537,Z 554.438,A 0.000,B 0.000,C 90.000,E1 294.771} C_DIS
LIN {X -0.351,Y -651.059,Z 554.435,A 0.000,B 0.000,C 90.000,E1 294.335} C_DIS
LIN {X -0.300,Y -649.185,Z 554.434,A 0.000,B 0.000,C 90.000,E1 294.207} C_DIS
LIN {X 0.099,Y -641.864,Z 554.432,A 0.000,B 0.000,C 90.000,E1 293.770} C_DIS
LIN {X -0.018,Y -639.938,Z 554.432,A 0.000,B 0.000,C 90.000,E1 293.695} C_DIS
LIN {X -0.183,Y -635.713,Z 554.431,A 0.000,B 0.000,C 90.000,E1 293.567} C_DIS
LIN {X -0.229,Y -634.614,Z 554.431,A 0.000,B 0.000,C 90.000,E1 293.515} C_DIS
LIN {X -0.056,Y -630.277,Z 554.430,A 0.000,B 0.000,C 90.000,E1 293.334} C_DIS
LIN {X -0.232,Y -620.528,Z 554.428,A 0.000,B 0.000,C 90.000,E1 293.025} C_DIS
LIN {X 0.112,Y -609.687,Z 554.426,A 0.000,B 0.000,C 90.000,E1 292.642} C_DIS
LIN {X -0.295,Y -588.819,Z 554.422,A 0.000,B 0.000,C 90.000,E1 292.025} C_DIS
LIN {X -0.082,Y -580.821,Z 554.421,A 0.000,B 0.000,C 90.000,E1 291.716} C_DIS
LIN {X 0.132,Y -574.449,Z 554.419,A 0.000,B 0.000,C 90.000,E1 291.408} C_DIS
LIN {X -0.085,Y -570.060,Z 554.418,A 0.000,B 0.000,C 90.000,E1 291.153} C_DIS
LIN {X 0.258,Y -568.650,Z 554.416,A 0.000,B 0.000,C 90.000,E1 290.918} C_DIS
LIN {X -0.173,Y -568.275,Z 554.415,A 0.000,B 0.000,C 90.000,E1 290.791} C_DIS
LIN {X -0.060,Y -568.044,Z 554.414,A 0.000,B 0.000,C 90.000,E1 290.556} C_DIS
LIN {X -0.153,Y -567.882,Z 554.404,A 0.000,B 0.000,C 90.000,E1 288.652} C_DIS
LIN {X 0.288,Y -567.695,Z 554.398,A 0.000,B 0.000,C 90.000,E1 287.511} C_DIS
LIN {X 0.188,Y -567.256,Z 554.390,A 0.000,B 0.000,C 90.000,E1 286.150} C_DIS
LIN {X -0.138,Y -566.398,Z 554.381,A 0.000,B 0.000,C 90.000,E1 284.537} C_DIS
LIN {X -0.088,Y -565.444,Z 554.372,A 0.000,B 0.000,C 90.000,E1 282.883} C_DIS
LIN {X -0.020,Y -564.382,Z 554.361,A 0.000,B 0.000,C 90.000,E1 280.950} C_DIS
LIN {X -0.019,Y -563.242,Z 554.349,A 0.000,B 0.000,C 90.000,E1 278.746} C_DIS
LIN {X -0.202,Y -562.364,Z 554.338,A 0.000,B 0.000,C 90.000,E1 276.834} C_DIS
LIN {X 0.260,Y -561.894,Z 554.332,A 0.000,B 0.000,C 90.000,E1 275.682} C_DIS
LIN {X 0.155,Y -561.474,Z 554.326,A 0.000,B 0.000,C 90.000,E1 274.588} C_DIS
LIN {X 0.216,Y -560.789,Z 554.316,A 0.000,B 0.000,C 90.000,E1 272.922} C_DIS
LIN {X -0.234,Y -559.938,Z 554.306,A 0.000,B 0.000,C 90.000,E1 271.031} C_DIS
LIN {X -0.243,Y -559.014,Z 554.296,A 0.000,B 0.000,C 90.000,E1 269.370} C_DIS
LIN {X -0.260,Y -558.125,Z 554.287,A 0.000,B 0.000,C 90.000,E1 267.707} C_DIS
LIN {X 0.255,Y -557.122,Z 554.278,A 0.000,B 0.000,C 90.000,E1 265.988} C_DIS
LIN {X 0.147,Y -556.266,Z 554.270,A 0.000,B 0.000,C 90.000,E1 264.609} C_DIS
LIN {X 0.207,Y -555.159,Z 554.261,A 0.000,B 0.000,C 90.000,E1 262.932} C_DIS
LIN {X 0.129,Y -554.114,Z 554.253,A 0.000,B 0.000,C 90.000,E1 261.546} C_DIS
LIN {X -0.010,Y -552.939,Z 554.247,A 0.000,B 0.000,C 90.000,E1 260.443} C_DIS
LIN {X -0.248,Y -550.287,Z 554.234,A 0.000,B 0.000,C 90.000,E1 258.229} C_DIS
LIN {X -0.005,Y -548.401,Z 554.225,A 0.000,B 0.000,C 90.000,E1 256.520} C_DIS
LIN {X 0.196,Y -546.277,Z 554.216,A 0.000,B 0.000,C 90.000,E1 254.810} C_DIS
LIN {X 0.083,Y -545.120,Z 554.211,A 0.000,B 0.000,C 90.000,E1 253.976} C_DIS
LIN {X 0.266,Y -542.941,Z 554.203,A 0.000,B 0.000,C 90.000,E1 252.543} C_DIS
LIN {X -0.173,Y -541.121,Z 554.197,A 0.000,B 0.000,C 90.000,E1 251.456} C_DIS
LIN {X 0.094,Y -538.662,Z 554.189,A 0.000,B 0.000,C 90.000,E1 250.007} C_DIS
LIN {X -0.007,Y -535.865,Z 554.181,A 0.000,B 0.000,C 90.000,E1 248.592} C_DIS
LIN {X -0.159,Y -532.880,Z 554.173,A 0.000,B 0.000,C 90.000,E1 247.177} C_DIS
LIN {X 0.133,Y -530.358,Z 554.167,A 0.000,B 0.000,C 90.000,E1 245.997} C_DIS
LIN {X 0.124,Y -527.645,Z 554.160,A 0.000,B 0.000,C 90.000,E1 244.845} C_DIS
LIN {X 0.246,Y -524.041,Z 554.152,A 0.000,B 0.000,C 90.000,E1 243.384} C_DIS
LIN {X -0.171,Y -520.242,Z 554.144,A 0.000,B 0.000,C 90.000,E1 241.975} C_DIS
LIN {X 0.291,Y -516.467,Z 554.136,A 0.000,B 0.000,C 90.000,E1 240.461} C_DIS
LIN {X -0.118,Y -513.183,Z 554.130,A 0.000,B 0.000,C 90.000,E1 239.331} C_DIS
LIN {X 0.097,Y -507.728,Z 554.120,A 0.000,B 0.000,C 90.000,E1 237.533} C_DIS
LIN {X -0.089,Y -501.611,Z 554.108,A 0.000,B 0.000,C 90.000,E1 235.468} C_DIS
LIN {X 0.010,Y -494.812,Z 554.095,A 0.000,B 0.000,C 90.000,E1 233.050} C_DIS
LIN {X -0.015,Y -490.709,Z 554.086,A 0.000,B 0.000,C 90.000,E1 231.537} C_DIS
LIN {X 0.152,Y -485.131,Z 554.074,A 0.000,B 0.000,C 90.000,E1 229.380} C_DIS
LIN {X -0.006,Y -480.378,Z 554.064,A 0.000,B 0.000,C 90.000,E1 227.553} C_DIS
LIN {X -0.187,Y -474.988,Z 554.052,A 0.000,B 0.000,C 90.000,E1 225.405} C_DIS
LIN {X -0.014,Y -471.306,Z 554.044,A 0.000,B 0.000,C 90.000,E1 223.824} C_DIS
LIN {X 0.232,Y -466.150,Z 554.031,A 0.000,B 0.000,C 90.000,E1 221.595} C_DIS
LIN {X 0.011,Y -461.815,Z 554.021,A 0.000,B 0.000,C 90.000,E1 219.725} C_DIS
LIN {X -0.047,Y -458.349,Z 554.012,A 0.000,B 0.000,C 90.000,E1 218.141} C_DIS
LIN {X -0.013,Y -454.187,Z 554.001,A 0.000,B 0.000,C 90.000,E1 216.217} C_DIS
LIN {X -0.046,Y -450.843,Z 553.992,A 0.000,B 0.000,C 90.000,E1 214.612} C_DIS
LIN {X -0.074,Y -446.932,Z 553.982,A 0.000,B 0.000,C 90.000,E1 212.673} C_DIS
LIN {X -0.005,Y -442.562,Z 553.969,A 0.000,B 0.000,C 90.000,E1 210.384} C_DIS
LIN {X 0.058,Y -438.945,Z 553.958,A 0.000,B 0.000,C 90.000,E1 208.409} C_DIS
LIN {X 0.036,Y -435.051,Z 553.945,A 0.000,B 0.000,C 90.000,E1 206.104} C_DIS
LIN {X 0.119,Y -431.231,Z 553.932,A 0.000,B 0.000,C 90.000,E1 203.770} C_DIS
LIN {X 0.114,Y -428.152,Z 553.921,A 0.000,B 0.000,C 90.000,E1 201.770} C_DIS
LIN {X -0.089,Y -424.813,Z 553.908,A 0.000,B 0.000,C 90.000,E1 199.450} C_DIS
LIN {X -0.080,Y -422.612,Z 553.899,A 0.000,B 0.000,C 90.000,E1 197.764} C_DIS
LIN {X -0.115,Y -420.444,Z 553.889,A 0.000,B 0.000,C 90.000,E1 196.079} C_DIS
LIN {X 0.142,Y -418.084,Z 553.878,A 0.000,B 0.000,C 90.000,E1 194.008} C_DIS
LIN {X 0.143,Y -416.275,Z 553.870,A 0.000,B 0.000,C 90.000,E1 192.647} C_DIS
LIN {X -0.138,Y -411.822,Z 553.851,A 0.000,B 0.000,C 90.000,E1 189.265} C_DIS
LIN {X 0.042,Y -408.837,Z 553.836,A 0.000,B 0.000,C 90.000,E1 186.486} C_DIS
LIN {X 0.010,Y -406.847,Z 553.825,A 0.000,B 0.000,C 90.000,E1 184.416} C_DIS
LIN {X -0.165,Y -404.020,Z 553.807,A 0.000,B 0.000,C 90.000,E1 181.318} C_DIS
LIN {X -0.094,Y -401.775,Z 553.788,A 0.000,B 0.000,C 90.000,E1 177.822} C_DIS
LIN {X 0.022,Y -400.600,Z 553.772,A 0.000,B 0.000,C 90.000,E1 175.008} C_DIS
LIN {X 0.150,Y -399.967,Z 553.755,A 0.000,B 0.000,C 90.000,E1 171.837} C_DIS
LIN {X 0.069,Y -399.891,Z 553.743,A 0.000,B 0.000,C 90.000,E1 169.746} C_DIS
LIN {X 0.111,Y -400.107,Z 553.728,A 0.000,B 0.000,C 90.000,E1 166.937} C_DIS
LIN {X -0.127,Y -400.654,Z 553.714,A 0.000,B 0.000,C 90.000,E1 164.519} C_DIS
LIN {X -0.022,Y -401.511,Z 553.700,A 0.000,B 0.000,C 90.000,E1 162.054} C_DIS
LIN {X -0.137,Y -402.606,Z 553.687,A 0.000,B 0.000,C 90.000,E1 159.625} C_DIS
LIN {X -0.181,Y -403.713,Z 553.675,A 0.000,B 0.000,C 90.000,E1 157.539} C_DIS
LIN {X -0.171,Y -405.133,Z 553.662,A 0.000,B 0.000,C 90.000,E1 155.101} C_DIS
LIN {X -0.045,Y -406.430,Z 553.650,A 0.000,B 0.000,C 90.000,E1 152.999} C_DIS
LIN {X -0.068,Y -407.644,Z 553.638,A 0.000,B 0.000,C 90.000,E1 150.923} C_DIS
LIN {X -0.138,Y -408.553,Z 553.629,A 0.000,B 0.000,C 90.000,E1 149.203} C_DIS
LIN {X 0.018,Y -409.250,Z 553.619,A 0.000,B 0.000,C 90.000,E1 147.454} C_DIS
LIN {X -0.011,Y -409.990,Z 553.608,A 0.000,B 0.000,C 90.000,E1 145.388} C_DIS
LIN {X 0.045,Y -410.374,Z 553.598,A 0.000,B 0.000,C 90.000,E1 143.657} C_DIS
LIN {X -0.058,Y -410.694,Z 553.589,A 0.000,B 0.000,C 90.000,E1 141.949} C_DIS
LIN {X 0.017,Y -410.828,Z 553.581,A 0.000,B 0.000,C 90.000,E1 140.561} C_DIS
LIN {X -0.066,Y -410.908,Z 553.571,A 0.000,B 0.000,C 90.000,E1 138.852} C_DIS
LIN {X -0.035,Y -410.936,Z 553.560,A 0.000,B 0.000,C 90.000,E1 136.782} C_DIS
LIN {X 0.119,Y -411.148,Z 553.547,A 0.000,B 0.000,C 90.000,E1 134.352} C_DIS
LIN {X 0.135,Y -411.336,Z 553.535,A 0.000,B 0.000,C 90.000,E1 132.285} C_DIS
LIN {X 0.162,Y -411.350,Z 553.527,A 0.000,B 0.000,C 90.000,E1 130.906} C_DIS
LIN {X 0.072,Y -411.247,Z 553.522,A 0.000,B 0.000,C 90.000,E1 129.886} C_DIS
LIN {X 0.247,Y -411.033,Z 553.516,A 0.000,B 0.000,C 90.000,E1 128.830} C_DIS
LIN {X 0.039,Y -410.545,Z 553.509,A 0.000,B 0.000,C 90.000,E1 127.649} C_DIS
LIN {X 0.001,Y -410.545,Z 553.509,A 0.000,B 0.000,C 90.000,E1 127.649} C_DIS
LIN {X 0.159,Y -415.095,Z 553.501,A 0.000,B 0.000,C 90.000,E1 126.091} C_DIS
LIN {X -0.247,Y -416.017,Z 553.499,A 0.000,B 0.000,C 90.000,E1 125.804} C_DIS
LIN {X 0.220,Y -425.525,Z 553.478,A 0.000,B 0.000,C 90.000,E1 122.005} C_DIS
LIN {X 0.164,Y -430.555,Z 553.469,A 0.000,B 0.000,C 90.000,E1 120.335} C_DIS
LIN {X -0.034,Y -441.467,Z 553.445,A 0.000,B 0.000,C 90.000,E1 116.052} C_DIS
LIN {X -0.116,Y -441.718,Z 553.444,A 0.000,B 0.000,C 90.000,E1 115.976} C_DIS
LIN {X -0.156,Y -441.821,Z 553.444,A 0.000,B 0.000,C 90.000,E1 115.976} C_DIS
LIN {X -0.185,Y -466.178,Z 553.438,A 0.000,B 0.000,C 90.000,E1 114.899} C_DIS
LIN {X -0.035,Y -481.830,Z 553.435,A 0.000,B 0.000,C 90.000,E1 114.207} C_DIS
LIN {X -0.018,Y -495.401,Z 553.431,A 0.000,B 0.000,C 90.000,E1 113.590} C_DIS
LIN {X 0.228,Y -505.425,Z 553.428,A 0.000,B 0.000,C 90.000,E1 113.078} C_DIS
LIN {X -0.206,Y -518.401,Z 553.425,A 0.000,B 0.000,C 90.000,E1 112.461} C_DIS
LIN {X -0.253,Y -526.512,Z 553.422,A 0.000,B 0.000,C 90.000,E1 112.025} C_DIS
LIN {X -0.132,Y -536.195,Z 553.419,A 0.000,B 0.000,C 90.000,E1 111.461} C_DIS
LIN {X -0.064,Y -543.936,Z 553.417,A 0.000,B 0.000,C 90.000,E1 110.972} C_DIS
LIN {X -0.049,Y -549.957,Z 553.414,A 0.000,B 0.000,C 90.000,E1 110.556} C_DIS
LIN {X -0.191,Y -554.392,Z 553.412,A 0.000,B 0.000,C 90.000,E1 110.248} C_DIS
LIN {X -0.106,Y -561.080,Z 553.409,A 0.000,B 0.000,C 90.000,E1 109.685} C_DIS
LIN {X -0.146,Y -563.581,Z 553.408,A 0.000,B 0.000,C 90.000,E1 109.450} C_DIS
LIN {X 0.175,Y -565.894,Z 553.407,A 0.000,B 0.000,C 90.000,E1 109.214} C_DIS
LIN {X 0.000,Y -569.495,Z 553.405,A 0.000,B 0.000,C 90.000,E1 108.852} C_DIS
LIN {X -0.086,Y -570.876,Z 553.404,A 0.000,B 0.000,C 90.000,E1 108.725} C_DIS
LIN {X 0.129,Y -574.205,Z 553.402,A 0.000,B 0.000,C 90.000,E1 108.308} C_DIS
LIN {X -0.050,Y -576.572,Z 553.400,A 0.000,B 0.000,C 90.000,E1 108.055} C_DIS
LIN {X -0.293,Y -581.707,Z 553.397,A 0.000,B 0.000,C 90.000,E1 107.402} C_DIS
LIN {X 0.115,Y -587.890,Z 553.391,A 0.000,B 0.000,C 90.000,E1 106.441} C_DIS
LIN {X 0.204,Y -591.298,Z 553.388,A 0.000,B 0.000,C 90.000,E1 105.898} C_DIS
LIN {X 0.084,Y -595.240,Z 553.385,A 0.000,B 0.000,C 90.000,E1 105.245} C_DIS
LIN {X -0.224,Y -599.508,Z 553.380,A 0.000,B 0.000,C 90.000,E1 104.481} C_DIS
LIN {X 0.243,Y -603.569,Z 553.376,A 0.000,B 0.000,C 90.000,E1 103.647} C_DIS
LIN {X -0.177,Y -608.173,Z 553.371,A 0.000,B 0.000,C 90.000,E1 102.771} C_DIS
LIN {X -0.164,Y -611.385,Z 553.367,A 0.000,B 0.000,C 90.000,E1 102.119} C_DIS
LIN {X 0.286,Y -614.985,Z 553.363,A 0.000,B 0.000,C 90.000,E1 101.299} C_DIS
LIN {X 0.052,Y -618.299,Z 553.359,A 0.000,B 0.000,C 90.000,E1 100.546} C_DIS
LIN {X 0.263,Y -627.438,Z 553.346,A 0.000,B 0.000,C 90.000,E1 98.219} C_DIS
LIN {X -0.142,Y -631.484,Z 553.340,A 0.000,B 0.000,C 90.000,E1 97.239} C_DIS
LIN {X 0.139,Y -635.328,Z 553.335,A 0.000,B 0.000,C 90.000,E1 96.201} C_DIS
LIN {X 0.300,Y -637.221,Z 553.332,A 0.000,B 0.000,C 90.000,E1 95.682} C_DIS
LIN {X 0.019,Y -640.559,Z 553.326,A 0.000,B 0.000,C 90.000,E1 94.702} C_DIS
LIN {X -0.034,Y -642.740,Z 553.322,A 0.000,B 0.000,C 90.000,E1 93.955} C_DIS
LIN {X -0.301,Y -645.411,Z 553.316,A 0.000,B 0.000,C 90.000,E1 92.980} C_DIS
LIN {X 0.086,Y -647.508,Z 553.311,A 0.000,B 0.000,C 90.000,E1 91.949} C_DIS
LIN {X 0.095,Y -648.770,Z 553.307,A 0.000,B 0.000,C 90.000,E1 91.203} C_DIS
LIN {X 0.099,Y -649.639,Z 553.303,A 0.000,B 0.000,C 90.000,E1 90.458} C_DIS
LIN {X 0.114,Y -650.298,Z 553.299,A 0.000,B 0.000,C 90.000,E1 89.714} C_DIS
LIN {X 0.134,Y -650.609,Z 553.294,A 0.000,B 0.000,C 90.000,E1 88.969} C_DIS
LIN {X -0.286,Y -650.630,Z 553.292,A 0.000,B 0.000,C 90.000,E1 88.511} C_DIS
LIN {X -0.245,Y -650.368,Z 553.288,A 0.000,B 0.000,C 90.000,E1 87.764} C_DIS
LIN {X -0.232,Y -649.868,Z 553.283,A 0.000,B 0.000,C 90.000,E1 87.020} C_DIS
LIN {X -0.194,Y -649.146,Z 553.279,A 0.000,B 0.000,C 90.000,E1 86.274} C_DIS
LIN {X -0.159,Y -648.149,Z 553.275,A 0.000,B 0.000,C 90.000,E1 85.527} C_DIS
LIN {X 0.340,Y -646.606,Z 553.270,A 0.000,B 0.000,C 90.000,E1 84.489} C_DIS
LIN {X -0.293,Y -645.128,Z 553.265,A 0.000,B 0.000,C 90.000,E1 83.799} C_DIS
LIN {X -0.060,Y -644.024,Z 553.263,A 0.000,B 0.000,C 90.000,E1 83.280} C_DIS
LIN {X -0.087,Y -642.062,Z 553.259,A 0.000,B 0.000,C 90.000,E1 82.534} C_DIS
LIN {X -0.224,Y -639.249,Z 553.253,A 0.000,B 0.000,C 90.000,E1 81.546} C_DIS
LIN {X -0.213,Y -636.839,Z 553.249,A 0.000,B 0.000,C 90.000,E1 80.792} C_DIS
LIN {X -0.227,Y -634.330,Z 553.245,A 0.000,B 0.000,C 90.000,E1 80.038} C_DIS
LIN {X 0.161,Y -630.673,Z 553.239,A 0.000,B 0.000,C 90.000,E1 78.993} C_DIS
LIN {X 0.198,Y -627.581,Z 553.235,A 0.000,B 0.000,C 90.000,E1 78.229} C_DIS
LIN {X 0.004,Y -623.231,Z 553.229,A 0.000,B 0.000,C 90.000,E1 77.229} C_DIS
LIN {X -0.025,Y -619.674,Z 553.225,A 0.000,B 0.000,C 90.000,E1 76.464} C_DIS
LIN {X 0.133,Y -617.140,Z 553.222,A 0.000,B 0.000,C 90.000,E1 75.936} C_DIS
LIN {X 0.030,Y -612.994,Z 553.218,A 0.000,B 0.000,C 90.000,E1 75.172} C_DIS
LIN {X 0.042,Y -608.532,Z 553.213,A 0.000,B 0.000,C 90.000,E1 74.393} C_DIS
LIN {X 0.024,Y -603.665,Z 553.209,A 0.000,B 0.000,C 90.000,E1 73.614} C_DIS
LIN {X 0.057,Y -598.346,Z 553.205,A 0.000,B 0.000,C 90.000,E1 72.851} C_DIS
LIN {X 0.223,Y -594.366,Z 553.202,A 0.000,B 0.000,C 90.000,E1 72.308} C_DIS
LIN {X 0.293,Y -588.717,Z 553.198,A 0.000,B 0.000,C 90.000,E1 71.638} C_DIS
LIN {X 0.015,Y -586.190,Z 553.197,A 0.000,B 0.000,C 90.000,E1 71.402} C_DIS
LIN {X -0.341,Y -582.603,Z 553.195,A 0.000,B 0.000,C 90.000,E1 71.040} C_DIS
LIN {X 0.107,Y -578.731,Z 553.192,A 0.000,B 0.000,C 90.000,E1 70.604} C_DIS
LIN {X -0.230,Y -571.969,Z 553.189,A 0.000,B 0.000,C 90.000,E1 70.007} C_DIS
LIN {X -0.065,Y -567.679,Z 553.187,A 0.000,B 0.000,C 90.000,E1 69.625} C_DIS
LIN {X 0.093,Y -563.331,Z 553.185,A 0.000,B 0.000,C 90.000,E1 69.263} C_DIS
LIN {X -0.068,Y -557.198,Z 553.182,A 0.000,B 0.000,C 90.000,E1 68.847} C_DIS
LIN {X -0.170,Y -552.307,Z 553.181,A 0.000,B 0.000,C 90.000,E1 68.539} C_DIS
LIN {X -0.201,Y -545.611,Z 553.179,A 0.000,B 0.000,C 90.000,E1 68.156} C_DIS
LIN {X 0.154,Y -540.589,Z 553.177,A 0.000,B 0.000,C 90.000,E1 67.847} C_DIS
LIN {X -0.054,Y -533.373,Z 553.175,A 0.000,B 0.000,C 90.000,E1 67.539} C_DIS
LIN {X 0.033,Y -526.323,Z 553.174,A 0.000,B 0.000,C 90.000,E1 67.230} C_DIS
LIN {X 0.139,Y -517.632,Z 553.172,A 0.000,B 0.000,C 90.000,E1 66.869} C_DIS
LIN {X 0.111,Y -501.460,Z 553.168,A 0.000,B 0.000,C 90.000,E1 66.305} C_DIS
LIN {X -0.051,Y -480.310,Z 553.165,A 0.000,B 0.000,C 90.000,E1 65.613} C_DIS
LIN {X -0.106,Y -460.963,Z 553.161,A 0.000,B 0.000,C 90.000,E1 64.921} C_DIS
LIN {X -0.139,Y -460.896,Z 553.161,A 0.000,B 0.000,C 90.000,E1 64.921} C_DIS
LIN {X 0.093,Y -455.619,Z 553.144,A 0.000,B 0.000,C 90.000,E1 61.975} C_DIS
LIN {X 0.081,Y -454.104,Z 553.141,A 0.000,B 0.000,C 90.000,E1 61.335} C_DIS
LIN {X 0.161,Y -445.092,Z 553.117,A 0.000,B 0.000,C 90.000,E1 57.120} C_DIS
LIN {X -0.089,Y -443.936,Z 553.114,A 0.000,B 0.000,C 90.000,E1 56.501} C_DIS
LIN {X -0.157,Y -440.587,Z 553.107,A 0.000,B 0.000,C 90.000,E1 55.182} C_DIS
LIN {X -0.197,Y -440.580,Z 553.106,A 0.000,B 0.000,C 90.000,E1 55.182} C_DIS
LIN {X -0.006,Y -443.060,Z 553.098,A 0.000,B 0.000,C 90.000,E1 53.543} C_DIS
LIN {X 0.000,Y -446.179,Z 553.087,A 0.000,B 0.000,C 90.000,E1 51.582} C_DIS
LIN {X 0.041,Y -448.064,Z 553.079,A 0.000,B 0.000,C 90.000,E1 50.275} C_DIS
LIN {X 0.092,Y -450.345,Z 553.070,A 0.000,B 0.000,C 90.000,E1 48.647} C_DIS
LIN {X -0.193,Y -452.527,Z 553.061,A 0.000,B 0.000,C 90.000,E1 47.067} C_DIS
LIN {X 0.193,Y -454.036,Z 553.054,A 0.000,B 0.000,C 90.000,E1 45.729} C_DIS
LIN {X -0.048,Y -455.184,Z 553.047,A 0.000,B 0.000,C 90.000,E1 44.474} C_DIS
LIN {X 0.008,Y -455.711,Z 553.044,A 0.000,B 0.000,C 90.000,E1 43.824} C_DIS
LIN {X 0.113,Y -456.386,Z 553.036,A 0.000,B 0.000,C 90.000,E1 42.528} C_DIS
LIN {X 0.251,Y -456.883,Z 553.029,A 0.000,B 0.000,C 90.000,E1 41.229} C_DIS
LIN {X -0.250,Y -457.139,Z 553.022,A 0.000,B 0.000,C 90.000,E1 40.011} C_DIS
LIN {X -0.042,Y -457.108,Z 553.015,A 0.000,B 0.000,C 90.000,E1 38.705} C_DIS
LIN {X 0.180,Y -456.944,Z 553.006,A 0.000,B 0.000,C 90.000,E1 37.076} C_DIS
LIN {X 0.109,Y -456.625,Z 552.999,A 0.000,B 0.000,C 90.000,E1 35.804} C_DIS
LIN {X 0.136,Y -456.011,Z 552.990,A 0.000,B 0.000,C 90.000,E1 34.199} C_DIS
LIN {X -0.101,Y -455.405,Z 552.981,A 0.000,B 0.000,C 90.000,E1 32.625} C_DIS
LIN {X 0.034,Y -454.875,Z 552.972,A 0.000,B 0.000,C 90.000,E1 31.003} C_DIS
LIN {X 0.023,Y -454.266,Z 552.962,A 0.000,B 0.000,C 90.000,E1 29.077} C_DIS
LIN {X 0.056,Y -453.522,Z 552.949,A 0.000,B 0.000,C 90.000,E1 26.821} C_DIS
LIN {X -0.129,Y -452.793,Z 552.937,A 0.000,B 0.000,C 90.000,E1 24.591} C_DIS
LIN {X -0.007,Y -452.347,Z 552.926,A 0.000,B 0.000,C 90.000,E1 22.642} C_DIS
LIN {X -0.245,Y -452.016,Z 552.915,A 0.000,B 0.000,C 90.000,E1 20.737} C_DIS
LIN {X -0.016,Y -451.735,Z 552.901,A 0.000,B 0.000,C 90.000,E1 18.127} C_DIS
LIN {X -0.070,Y -451.797,Z 552.886,A 0.000,B 0.000,C 90.000,E1 15.552} C_DIS
LIN {X -0.064,Y -452.259,Z 552.870,A 0.000,B 0.000,C 90.000,E1 12.647} C_DIS
LIN {X 0.125,Y -453.011,Z 552.858,A 0.000,B 0.000,C 90.000,E1 10.366} C_DIS
LIN {X -0.060,Y -454.232,Z 552.843,A 0.000,B 0.000,C 90.000,E1 7.814} C_DIS
LIN {X -0.085,Y -455.634,Z 552.831,A 0.000,B 0.000,C 90.000,E1 5.568} C_DIS
LIN {X -0.104,Y -457.219,Z 552.818,A 0.000,B 0.000,C 90.000,E1 3.326} C_DIS
LIN {X 0.019,Y -460.150,Z 552.801,A 0.000,B 0.000,C 90.000,E1 0.115} C_DIS
LIN {X 0.036,Y -462.709,Z 552.788,A 0.000,B 0.000,C 90.000,E1 357.879} C_DIS
LIN {X -0.061,Y -466.053,Z 552.774,A 0.000,B 0.000,C 90.000,E1 355.355} C_DIS
LIN {X -0.041,Y -467.799,Z 552.767,A 0.000,B 0.000,C 90.000,E1 354.090} C_DIS
LIN {X -0.129,Y -469.971,Z 552.758,A 0.000,B 0.000,C 90.000,E1 352.527} C_DIS
LIN {X -0.122,Y -472.996,Z 552.746,A 0.000,B 0.000,C 90.000,E1 350.330} C_DIS
LIN {X 0.110,Y -476.334,Z 552.734,A 0.000,B 0.000,C 90.000,E1 348.117} C_DIS
LIN {X 0.170,Y -479.862,Z 552.722,A 0.000,B 0.000,C 90.000,E1 345.936} C_DIS
LIN {X -0.001,Y -483.067,Z 552.712,A 0.000,B 0.000,C 90.000,E1 344.102} C_DIS
LIN {X 0.032,Y -487.137,Z 552.700,A 0.000,B 0.000,C 90.000,E1 341.945} C_DIS
LIN {X -0.031,Y -490.135,Z 552.691,A 0.000,B 0.000,C 90.000,E1 340.423} C_DIS
LIN {X 0.004,Y -493.698,Z 552.681,A 0.000,B 0.000,C 90.000,E1 338.592} C_DIS
LIN {X 0.191,Y -496.028,Z 552.674,A 0.000,B 0.000,C 90.000,E1 337.358} C_DIS
LIN {X 0.008,Y -498.851,Z 552.666,A 0.000,B 0.000,C 90.000,E1 335.869} C_DIS
LIN {X 0.076,Y -501.571,Z 552.658,A 0.000,B 0.000,C 90.000,E1 334.357} C_DIS
LIN {X -0.036,Y -504.211,Z 552.649,A 0.000,B 0.000,C 90.000,E1 332.871} C_DIS
LIN {X -0.095,Y -506.750,Z 552.641,A 0.000,B 0.000,C 90.000,E1 331.385} C_DIS
LIN {X 0.101,Y -510.345,Z 552.629,A 0.000,B 0.000,C 90.000,E1 329.282} C_DIS
LIN {X 0.224,Y -512.930,Z 552.621,A 0.000,B 0.000,C 90.000,E1 327.788} C_DIS
LIN {X 0.325,Y -516.056,Z 552.611,A 0.000,B 0.000,C 90.000,E1 326.008} C_DIS
LIN {X 0.122,Y -518.704,Z 552.603,A 0.000,B 0.000,C 90.000,E1 324.562} C_DIS
LIN {X -0.208,Y -521.762,Z 552.594,A 0.000,B 0.000,C 90.000,E1 322.844} C_DIS
LIN {X -0.188,Y -525.586,Z 552.582,A 0.000,B 0.000,C 90.000,E1 320.803} C_DIS
LIN {X 0.069,Y -532.282,Z 552.565,A 0.000,B 0.000,C 90.000,E1 317.595} C_DIS
LIN {X 0.255,Y -537.008,Z 552.553,A 0.000,B 0.000,C 90.000,E1 315.567} C_DIS
LIN {X -0.220,Y -541.967,Z 552.542,A 0.000,B 0.000,C 90.000,E1 313.623} C_DIS
LIN {X 0.211,Y -547.148,Z 552.531,A 0.000,B 0.000,C 90.000,E1 311.595} C_DIS
LIN {X -0.088,Y -549.289,Z 552.527,A 0.000,B 0.000,C 90.000,E1 310.782} C_DIS
LIN {X -0.107,Y -551.499,Z 552.522,A 0.000,B 0.000,C 90.000,E1 310.011} C_DIS
LIN {X -0.119,Y -553.412,Z 552.520,A 0.000,B 0.000,C 90.000,E1 309.564} C_DIS
LIN {X -0.015,Y -553.688,Z 552.519,A 0.000,B 0.000,C 90.000,E1 309.483} C_DIS
LIN {X -0.057,Y -555.211,Z 552.518,A 0.000,B 0.000,C 90.000,E1 309.277} C_DIS
LIN {X 0.013,Y -556.839,Z 552.517,A 0.000,B 0.000,C 90.000,E1 308.991} C_DIS
LIN {X 0.092,Y -558.894,Z 552.515,A 0.000,B 0.000,C 90.000,E1 308.705} C_DIS
LIN {X -0.028,Y -562.661,Z 552.513,A 0.000,B 0.000,C 90.000,E1 308.302} C_DIS
LIN {X -0.043,Y -566.272,Z 552.511,A 0.000,B 0.000,C 90.000,E1 307.971} C_DIS
LIN {X -0.221,Y -571.991,Z 552.508,A 0.000,B 0.000,C 90.000,E1 307.523} C_DIS
LIN {X -0.327,Y -580.474,Z 552.505,A 0.000,B 0.000,C 90.000,E1 306.870} C_DIS
LIN {X -0.098,Y -584.648,Z 552.503,A 0.000,B 0.000,C 90.000,E1 306.503} C_DIS
LIN {X 0.050,Y -588.678,Z 552.501,A 0.000,B 0.000,C 90.000,E1 306.137} C_DIS
LIN {X 0.066,Y -593.847,Z 552.498,A 0.000,B 0.000,C 90.000,E1 305.644} C_DIS
LIN {X 0.057,Y -597.608,Z 552.496,A 0.000,B 0.000,C 90.000,E1 305.264} C_DIS
LIN {X -0.116,Y -607.223,Z 552.490,A 0.000,B 0.000,C 90.000,E1 304.246} C_DIS
LIN {X 0.040,Y -614.317,Z 552.486,A 0.000,B 0.000,C 90.000,E1 303.452} C_DIS
LIN {X 0.124,Y -622.338,Z 552.481,A 0.000,B 0.000,C 90.000,E1 302.546} C_DIS
LIN {X -0.091,Y -629.842,Z 552.476,A 0.000,B 0.000,C 90.000,E1 301.671} C_DIS
LIN {X 0.273,Y -633.763,Z 552.473,A 0.000,B 0.000,C 90.000,E1 301.131} C_DIS
LIN {X -0.186,Y -638.003,Z 552.470,A 0.000,B 0.000,C 90.000,E1 300.541} C_DIS
LIN {X 0.265,Y -641.631,Z 552.466,A 0.000,B 0.000,C 90.000,E1 299.873} C_DIS
LIN {X -0.132,Y -644.605,Z 552.463,A 0.000,B 0.000,C 90.000,E1 299.283} C_DIS
LIN {X -0.161,Y -647.477,Z 552.458,A 0.000,B 0.000,C 90.000,E1 298.537} C_DIS
LIN {X -0.094,Y -653.629,Z 552.449,A 0.000,B 0.000,C 90.000,E1 296.796} C_DIS
LIN {X 0.011,Y -654.530,Z 552.448,A 0.000,B 0.000,C 90.000,E1 296.539} C_DIS
LIN {X 0.118,Y -655.082,Z 552.446,A 0.000,B 0.000,C 90.000,E1 296.283} C_DIS
LIN {X 0.057,Y -655.653,Z 552.443,A 0.000,B 0.000,C 90.000,E1 295.796} C_DIS
LIN {X 0.173,Y -655.486,Z 552.442,A 0.000,B 0.000,C 90.000,E1 295.540} C_DIS
LIN {X -0.190,Y -654.280,Z 552.439,A 0.000,B 0.000,C 90.000,E1 295.079} C_DIS
LIN {X -0.079,Y -653.050,Z 552.438,A 0.000,B 0.000,C 90.000,E1 294.823} C_DIS
LIN {X -0.243,Y -651.023,Z 552.437,A 0.000,B 0.000,C 90.000,E1 294.591} C_DIS
LIN {X -0.192,Y -649.928,Z 552.436,A 0.000,B 0.000,C 90.000,E1 294.463} C_DIS
LIN {X -0.141,Y -648.561,Z 552.435,A 0.000,B 0.000,C 90.000,E1 294.335} C_DIS
LIN {X 0.119,Y -644.307,Z 552.434,A 0.000,B 0.000,C 90.000,E1 294.079} C_DIS
LIN {X 0.255,Y -642.196,Z 552.433,A 0.000,B 0.000,C 90.000,E1 293.898} C_DIS
LIN {X -0.164,Y -638.995,Z 552.432,A 0.000,B 0.000,C 90.000,E1 293.770} C_DIS
LIN {X -0.224,Y -636.899,Z 552.432,A 0.000,B 0.000,C 90.000,E1 293.695} C_DIS
LIN {X -0.056,Y -633.507,Z 552.431,A 0.000,B 0.000,C 90.000,E1 293.515} C_DIS
LIN {X 0.330,Y -618.861,Z 552.428,A 0.000,B 0.000,C 90.000,E1 292.950} C_DIS
LIN {X 0.128,Y -601.504,Z 552.425,A 0.000,B 0.000,C 90.000,E1 292.408} C_DIS
LIN {X 0.031,Y -587.605,Z 552.422,A 0.000,B 0.000,C 90.000,E1 291.972} C_DIS
LIN {X 0.280,Y -581.156,Z 552.421,A 0.000,B 0.000,C 90.000,E1 291.716} C_DIS
LIN {X -0.280,Y -575.902,Z 552.420,A 0.000,B 0.000,C 90.000,E1 291.535} C_DIS
LIN {X 0.179,Y -573.436,Z 552.419,A 0.000,B 0.000,C 90.000,E1 291.354} C_DIS
LIN {X 0.083,Y -571.284,Z 552.418,A 0.000,B 0.000,C 90.000,E1 291.227} C_DIS
LIN {X 0.099,Y -570.383,Z 552.418,A 0.000,B 0.000,C 90.000,E1 291.153} C_DIS
LIN {X -0.171,Y -569.020,Z 552.416,A 0.000,B 0.000,C 90.000,E1 290.972} C_DIS
LIN {X -0.223,Y -569.005,Z 552.416,A 0.000,B 0.000,C 90.000,E1 290.972} C_DIS
LIN {X -0.137,Y -568.601,Z 552.415,A 0.000,B 0.000,C 90.000,E1 290.663} C_DIS
LIN {X 0.171,Y -568.453,Z 552.404,A 0.000,B 0.000,C 90.000,E1 288.725} C_DIS
LIN {X -0.292,Y -568.197,Z 552.397,A 0.000,B 0.000,C 90.000,E1 287.402} C_DIS
LIN {X 0.159,Y -567.843,Z 552.391,A 0.000,B 0.000,C 90.000,E1 286.260} C_DIS
LIN {X 0.071,Y -567.190,Z 552.383,A 0.000,B 0.000,C 90.000,E1 284.898} C_DIS
LIN {X -0.198,Y -566.536,Z 552.377,A 0.000,B 0.000,C 90.000,E1 283.828} C_DIS
LIN {X 0.234,Y -565.740,Z 552.369,A 0.000,B 0.000,C 90.000,E1 282.411} C_DIS
LIN {X 0.030,Y -564.847,Z 552.360,A 0.000,B 0.000,C 90.000,E1 280.782} C_DIS
LIN {X 0.142,Y -563.762,Z 552.348,A 0.000,B 0.000,C 90.000,E1 278.568} C_DIS
LIN {X -0.107,Y -562.894,Z 552.337,A 0.000,B 0.000,C 90.000,E1 276.663} C_DIS
LIN {X 0.277,Y -562.550,Z 552.332,A 0.000,B 0.000,C 90.000,E1 275.796} C_DIS
LIN {X 0.272,Y -561.993,Z 552.325,A 0.000,B 0.000,C 90.000,E1 274.416} C_DIS
LIN {X 0.252,Y -561.435,Z 552.317,A 0.000,B 0.000,C 90.000,E1 273.037} C_DIS
LIN {X -0.184,Y -560.560,Z 552.306,A 0.000,B 0.000,C 90.000,E1 271.146} C_DIS
LIN {X -0.090,Y -559.429,Z 552.296,A 0.000,B 0.000,C 90.000,E1 269.198} C_DIS
LIN {X -0.185,Y -558.681,Z 552.288,A 0.000,B 0.000,C 90.000,E1 267.822} C_DIS
LIN {X -0.212,Y -557.667,Z 552.279,A 0.000,B 0.000,C 90.000,E1 266.159} C_DIS
LIN {X 0.248,Y -556.825,Z 552.271,A 0.000,B 0.000,C 90.000,E1 264.723} C_DIS
LIN {X 0.254,Y -555.699,Z 552.262,A 0.000,B 0.000,C 90.000,E1 263.053} C_DIS
LIN {X -0.247,Y -554.396,Z 552.252,A 0.000,B 0.000,C 90.000,E1 261.432} C_DIS
LIN {X 0.130,Y -553.516,Z 552.248,A 0.000,B 0.000,C 90.000,E1 260.557} C_DIS
LIN {X -0.086,Y -550.852,Z 552.235,A 0.000,B 0.000,C 90.000,E1 258.342} C_DIS
LIN {X 0.049,Y -548.943,Z 552.226,A 0.000,B 0.000,C 90.000,E1 256.645} C_DIS
LIN {X 0.061,Y -547.497,Z 552.220,A 0.000,B 0.000,C 90.000,E1 255.519} C_DIS
LIN {X 0.055,Y -546.038,Z 552.213,A 0.000,B 0.000,C 90.000,E1 254.393} C_DIS
LIN {X 0.020,Y -544.347,Z 552.207,A 0.000,B 0.000,C 90.000,E1 253.268} C_DIS
LIN {X -0.107,Y -541.588,Z 552.198,A 0.000,B 0.000,C 90.000,E1 251.583} C_DIS
LIN {X 0.166,Y -539.127,Z 552.190,A 0.000,B 0.000,C 90.000,E1 250.134} C_DIS
LIN {X -0.147,Y -536.909,Z 552.183,A 0.000,B 0.000,C 90.000,E1 249.028} C_DIS
LIN {X -0.077,Y -533.977,Z 552.176,A 0.000,B 0.000,C 90.000,E1 247.592} C_DIS
LIN {X 0.029,Y -531.481,Z 552.169,A 0.000,B 0.000,C 90.000,E1 246.433} C_DIS
LIN {X 0.035,Y -528.819,Z 552.163,A 0.000,B 0.000,C 90.000,E1 245.281} C_DIS
LIN {X -0.214,Y -525.990,Z 552.156,A 0.000,B 0.000,C 90.000,E1 244.152} C_DIS
LIN {X -0.276,Y -522.987,Z 552.150,A 0.000,B 0.000,C 90.000,E1 242.999} C_DIS
LIN {X -0.008,Y -519.179,Z 552.142,A 0.000,B 0.000,C 90.000,E1 241.513} C_DIS
LIN {X 0.070,Y -516.084,Z 552.135,A 0.000,B 0.000,C 90.000,E1 240.333} C_DIS
LIN {X 0.004,Y -513.647,Z 552.130,A 0.000,B 0.000,C 90.000,E1 239.459} C_DIS
LIN {X 0.232,Y -508.229,Z 552.121,A 0.000,B 0.000,C 90.000,E1 237.661} C_DIS
LIN {X 0.061,Y -502.041,Z 552.109,A 0.000,B 0.000,C 90.000,E1 235.595} C_DIS
LIN {X 0.149,Y -496.924,Z 552.099,A 0.000,B 0.000,C 90.000,E1 233.783} C_DIS
LIN {X -0.139,Y -491.141,Z 552.087,A 0.000,B 0.000,C 90.000,E1 231.698} C_DIS
LIN {X 0.036,Y -485.521,Z 552.075,A 0.000,B 0.000,C 90.000,E1 229.542} C_DIS
LIN {X -0.115,Y -480.772,Z 552.065,A 0.000,B 0.000,C 90.000,E1 227.715} C_DIS
LIN {X -0.178,Y -474.584,Z 552.051,A 0.000,B 0.000,C 90.000,E1 225.243} C_DIS
LIN {X -0.013,Y -470.875,Z 552.043,A 0.000,B 0.000,C 90.000,E1 223.662} C_DIS
LIN {X 0.152,Y -466.471,Z 552.032,A 0.000,B 0.000,C 90.000,E1 221.757} C_DIS
LIN {X 0.191,Y -462.870,Z 552.023,A 0.000,B 0.000,C 90.000,E1 220.172} C_DIS
LIN {X -0.105,Y -458.653,Z 552.013,A 0.000,B 0.000,C 90.000,E1 218.302} C_DIS
LIN {X 0.214,Y -455.191,Z 552.004,A 0.000,B 0.000,C 90.000,E1 216.664} C_DIS
LIN {X 0.178,Y -451.121,Z 551.993,A 0.000,B 0.000,C 90.000,E1 214.739} C_DIS
LIN {X -0.091,Y -447.206,Z 551.982,A 0.000,B 0.000,C 90.000,E1 212.832} C_DIS
LIN {X -0.004,Y -442.790,Z 551.970,A 0.000,B 0.000,C 90.000,E1 210.541} C_DIS
LIN {X 0.076,Y -439.203,Z 551.959,A 0.000,B 0.000,C 90.000,E1 208.565} C_DIS
LIN {X 0.092,Y -434.684,Z 551.944,A 0.000,B 0.000,C 90.000,E1 205.924} C_DIS
LIN {X -0.040,Y -431.424,Z 551.933,A 0.000,B 0.000,C 90.000,E1 203.951} C_DIS
LIN {X -0.042,Y -428.349,Z 551.922,A 0.000,B 0.000,C 90.000,E1 201.950} C_DIS
LIN {X 0.143,Y -424.106,Z 551.905,A 0.000,B 0.000,C 90.000,E1 198.906} C_DIS
LIN {X 0.138,Y -421.877,Z 551.896,A 0.000,B 0.000,C 90.000,E1 197.221} C_DIS
LIN {X -0.031,Y -419.761,Z 551.886,A 0.000,B 0.000,C 90.000,E1 195.552} C_DIS
LIN {X 0.161,Y -417.844,Z 551.877,A 0.000,B 0.000,C 90.000,E1 193.828} C_DIS
LIN {X 0.065,Y -415.996,Z 551.869,A 0.000,B 0.000,C 90.000,E1 192.479} C_DIS
LIN {X 0.186,Y -412.435,Z 551.854,A 0.000,B 0.000,C 90.000,E1 189.726} C_DIS
LIN {X -0.025,Y -409.385,Z 551.839,A 0.000,B 0.000,C 90.000,E1 187.004} C_DIS
LIN {X -0.034,Y -407.049,Z 551.826,A 0.000,B 0.000,C 90.000,E1 184.588} C_DIS
LIN {X -0.176,Y -404.512,Z 551.810,A 0.000,B 0.000,C 90.000,E1 181.833} C_DIS
LIN {X -0.062,Y -402.309,Z 551.793,A 0.000,B 0.000,C 90.000,E1 178.682} C_DIS
LIN {X 0.065,Y -401.004,Z 551.777,A 0.000,B 0.000,C 90.000,E1 175.869} C_DIS
LIN {X 0.168,Y -400.162,Z 551.760,A 0.000,B 0.000,C 90.000,E1 172.704} C_DIS
LIN {X 0.042,Y -400.006,Z 551.750,A 0.000,B 0.000,C 90.000,E1 170.971} C_DIS
LIN {X 0.044,Y -400.007,Z 551.740,A 0.000,B 0.000,C 90.000,E1 169.218} C_DIS
LIN {X 0.093,Y -400.339,Z 551.725,A 0.000,B 0.000,C 90.000,E1 166.408} C_DIS
LIN {X 0.050,Y -401.083,Z 551.709,A 0.000,B 0.000,C 90.000,E1 163.614} C_DIS
LIN {X 0.176,Y -401.989,Z 551.695,A 0.000,B 0.000,C 90.000,E1 161.148} C_DIS
LIN {X -0.023,Y -403.018,Z 551.684,A 0.000,B 0.000,C 90.000,E1 159.082} C_DIS
LIN {X 0.091,Y -404.142,Z 551.672,A 0.000,B 0.000,C 90.000,E1 156.975} C_DIS
LIN {X -0.145,Y -405.427,Z 551.661,A 0.000,B 0.000,C 90.000,E1 154.921} C_DIS
LIN {X -0.018,Y -406.726,Z 551.649,A 0.000,B 0.000,C 90.000,E1 152.820} C_DIS
LIN {X 0.244,Y -407.757,Z 551.639,A 0.000,B 0.000,C 90.000,E1 151.051} C_DIS
LIN {X 0.178,Y -408.683,Z 551.630,A 0.000,B 0.000,C 90.000,E1 149.331} C_DIS
LIN {X -0.084,Y -409.583,Z 551.618,A 0.000,B 0.000,C 90.000,E1 147.296} C_DIS
LIN {X -0.098,Y -410.288,Z 551.607,A 0.000,B 0.000,C 90.000,E1 145.229} C_DIS
LIN {X -0.031,Y -410.673,Z 551.597,A 0.000,B 0.000,C 90.000,E1 143.497} C_DIS
LIN {X -0.054,Y -410.983,Z 551.588,A 0.000,B 0.000,C 90.000,E1 141.778} C_DIS
LIN {X -0.039,Y -411.104,Z 551.580,A 0.000,B 0.000,C 90.000,E1 140.400} C_DIS
LIN {X -0.115,Y -411.184,Z 551.570,A 0.000,B 0.000,C 90.000,E1 138.690} C_DIS
LIN {X -0.076,Y -411.226,Z 551.559,A 0.000,B 0.000,C 90.000,E1 136.620} C_DIS
LIN {X 0.088,Y -411.441,Z 551.546,A 0.000,B 0.000,C 90.000,E1 134.190} C_DIS
LIN {X 0.108,Y -411.584,Z 551.534,A 0.000,B 0.000,C 90.000,E1 132.123} C_DIS
LIN {X -0.131,Y -411.541,Z 551.526,A 0.000,B 0.000,C 90.000,E1 130.782} C_DIS
LIN {X 0.049,Y -411.437,Z 551.521,A 0.000,B 0.000,C 90.000,E1 129.725} C_DIS
LIN {X -0.033,Y -411.167,Z 551.515,A 0.000,B 0.000,C 90.000,E1 128.705} C_DIS
LIN {X 0.037,Y -410.676,Z 551.509,A 0.000,B 0.000,C 90.000,E1 127.604} C_DIS
LIN {X -0.002,Y -410.675,Z 551.509,A 0.000,B 0.000,C 90.000,E1 127.604} C_DIS
LIN {X 0.137,Y -415.594,Z 551.500,A 0.000,B 0.000,C 90.000,E1 125.931} C_DIS
LIN {X -0.024,Y -425.985,Z 551.477,A 0.000,B 0.000,C 90.000,E1 121.878} C_DIS
LIN {X -0.071,Y -430.982,Z 551.468,A 0.000,B 0.000,C 90.000,E1 120.207} C_DIS
LIN {X 0.075,Y -440.047,Z 551.448,A 0.000,B 0.000,C 90.000,E1 116.539} C_DIS
LIN {X -0.055,Y -442.592,Z 551.443,A 0.000,B 0.000,C 90.000,E1 115.668} C_DIS
LIN {X -0.095,Y -442.689,Z 551.443,A 0.000,B 0.000,C 90.000,E1 115.668} C_DIS
LIN {X 0.087,Y -465.568,Z 551.437,A 0.000,B 0.000,C 90.000,E1 114.643} C_DIS
LIN {X 0.092,Y -482.962,Z 551.433,A 0.000,B 0.000,C 90.000,E1 113.898} C_DIS
LIN {X -0.319,Y -496.524,Z 551.430,A 0.000,B 0.000,C 90.000,E1 113.334} C_DIS
LIN {X 0.240,Y -503.230,Z 551.428,A 0.000,B 0.000,C 90.000,E1 112.950} C_DIS
LIN {X -0.026,Y -516.234,Z 551.424,A 0.000,B 0.000,C 90.000,E1 112.333} C_DIS
LIN {X 0.063,Y -524.332,Z 551.422,A 0.000,B 0.000,C 90.000,E1 111.897} C_DIS
LIN {X 0.064,Y -534.102,Z 551.419,A 0.000,B 0.000,C 90.000,E1 111.354} C_DIS
LIN {X -0.131,Y -538.835,Z 551.417,A 0.000,B 0.000,C 90.000,E1 111.099} C_DIS
LIN {X -0.290,Y -544.816,Z 551.415,A 0.000,B 0.000,C 90.000,E1 110.737} C_DIS
LIN {X 0.191,Y -547.938,Z 551.414,A 0.000,B 0.000,C 90.000,E1 110.482} C_DIS
LIN {X 0.165,Y -553.891,Z 551.412,A 0.000,B 0.000,C 90.000,E1 110.066} C_DIS
LIN {X 0.066,Y -559.486,Z 551.409,A 0.000,B 0.000,C 90.000,E1 109.631} C_DIS
LIN {X 0.037,Y -565.630,Z 551.406,A 0.000,B 0.000,C 90.000,E1 109.087} C_DIS
LIN {X 0.190,Y -570.379,Z 551.404,A 0.000,B 0.000,C 90.000,E1 108.598} C_DIS
LIN {X -0.014,Y -576.343,Z 551.400,A 0.000,B 0.000,C 90.000,E1 107.946} C_DIS
LIN {X -0.001,Y -580.658,Z 551.397,A 0.000,B 0.000,C 90.000,E1 107.402} C_DIS
LIN {X -0.292,Y -586.249,Z 551.392,A 0.000,B 0.000,C 90.000,E1 106.622} C_DIS
LIN {X 0.275,Y -590.670,Z 551.389,A 0.000,B 0.000,C 90.000,E1 105.898} C_DIS
LIN {X 0.150,Y -594.747,Z 551.385,A 0.000,B 0.000,C 90.000,E1 105.245} C_DIS
LIN {X 0.153,Y -599.666,Z 551.380,A 0.000,B 0.000,C 90.000,E1 104.356} C_DIS
LIN {X -0.108,Y -603.829,Z 551.375,A 0.000,B 0.000,C 90.000,E1 103.592} C_DIS
LIN {X 0.264,Y -607.911,Z 551.371,A 0.000,B 0.000,C 90.000,E1 102.771} C_DIS
LIN {X 0.197,Y -611.839,Z 551.367,A 0.000,B 0.000,C 90.000,E1 102.007} C_DIS
LIN {X -0.128,Y -616.071,Z 551.362,A 0.000,B 0.000,C 90.000,E1 101.130} C_DIS
LIN {X -0.240,Y -619.335,Z 551.358,A 0.000,B 0.000,C 90.000,E1 100.366} C_DIS
LIN {X -0.101,Y -628.640,Z 551.345,A 0.000,B 0.000,C 90.000,E1 98.049} C_DIS
LIN {X 0.142,Y -632.697,Z 551.339,A 0.000,B 0.000,C 90.000,E1 97.011} C_DIS
LIN {X 0.246,Y -637.560,Z 551.332,A 0.000,B 0.000,C 90.000,E1 95.739} C_DIS
LIN {X -0.031,Y -640.928,Z 551.326,A 0.000,B 0.000,C 90.000,E1 94.759} C_DIS
LIN {X -0.082,Y -643.178,Z 551.322,A 0.000,B 0.000,C 90.000,E1 94.012} C_DIS
LIN {X 0.300,Y -645.902,Z 551.317,A 0.000,B 0.000,C 90.000,E1 92.980} C_DIS
LIN {X 0.049,Y -648.046,Z 551.311,A 0.000,B 0.000,C 90.000,E1 92.007} C_DIS
LIN {X 0.063,Y -649.364,Z 551.307,A 0.000,B 0.000,C 90.000,E1 91.260} C_DIS
LIN {X 0.073,Y -650.260,Z 551.303,A 0.000,B 0.000,C 90.000,E1 90.516} C_DIS
LIN {X 0.094,Y -650.916,Z 551.299,A 0.000,B 0.000,C 90.000,E1 89.771} C_DIS
LIN {X -0.323,Y -651.159,Z 551.296,A 0.000,B 0.000,C 90.000,E1 89.312} C_DIS
LIN {X -0.296,Y -651.288,Z 551.292,A 0.000,B 0.000,C 90.000,E1 88.568} C_DIS
LIN {X -0.248,Y -651.049,Z 551.288,A 0.000,B 0.000,C 90.000,E1 87.822} C_DIS
LIN {X -0.228,Y -650.532,Z 551.284,A 0.000,B 0.000,C 90.000,E1 87.078} C_DIS
LIN {X -0.182,Y -649.801,Z 551.280,A 0.000,B 0.000,C 90.000,E1 86.331} C_DIS
LIN {X -0.140,Y -648.823,Z 551.275,A 0.000,B 0.000,C 90.000,E1 85.584} C_DIS
LIN {X -0.337,Y -647.253,Z 551.270,A 0.000,B 0.000,C 90.000,E1 84.609} C_DIS
LIN {X -0.258,Y -645.750,Z 551.266,A 0.000,B 0.000,C 90.000,E1 83.856} C_DIS
LIN {X -0.020,Y -644.637,Z 551.263,A 0.000,B 0.000,C 90.000,E1 83.337} C_DIS
LIN {X -0.208,Y -641.954,Z 551.258,A 0.000,B 0.000,C 90.000,E1 82.356} C_DIS
LIN {X -0.169,Y -639.765,Z 551.253,A 0.000,B 0.000,C 90.000,E1 81.602} C_DIS
LIN {X 0.198,Y -636.500,Z 551.248,A 0.000,B 0.000,C 90.000,E1 80.566} C_DIS
LIN {X -0.159,Y -634.757,Z 551.245,A 0.000,B 0.000,C 90.000,E1 80.095} C_DIS
LIN {X 0.237,Y -631.016,Z 551.239,A 0.000,B 0.000,C 90.000,E1 79.050} C_DIS
LIN {X -0.144,Y -628.973,Z 551.237,A 0.000,B 0.000,C 90.000,E1 78.578} C_DIS
LIN {X -0.115,Y -625.679,Z 551.232,A 0.000,B 0.000,C 90.000,E1 77.813} C_DIS
LIN {X -0.293,Y -621.616,Z 551.227,A 0.000,B 0.000,C 90.000,E1 76.937} C_DIS
LIN {X 0.258,Y -617.856,Z 551.223,A 0.000,B 0.000,C 90.000,E1 76.117} C_DIS
LIN {X 0.119,Y -612.945,Z 551.218,A 0.000,B 0.000,C 90.000,E1 75.227} C_DIS
LIN {X 0.131,Y -608.366,Z 551.214,A 0.000,B 0.000,C 90.000,E1 74.448} C_DIS
LIN {X -0.067,Y -603.384,Z 551.209,A 0.000,B 0.000,C 90.000,E1 73.685} C_DIS
LIN {X 0.079,Y -598.768,Z 551.206,A 0.000,B 0.000,C 90.000,E1 73.015} C_DIS
LIN {X 0.012,Y -593.589,Z 551.202,A 0.000,B 0.000,C 90.000,E1 72.362} C_DIS
LIN {X 0.146,Y -589.009,Z 551.199,A 0.000,B 0.000,C 90.000,E1 71.819} C_DIS
LIN {X -0.221,Y -581.672,Z 551.195,A 0.000,B 0.000,C 90.000,E1 71.094} C_DIS
LIN {X 0.091,Y -577.716,Z 551.193,A 0.000,B 0.000,C 90.000,E1 70.678} C_DIS
LIN {X 0.050,Y -572.352,Z 551.190,A 0.000,B 0.000,C 90.000,E1 70.188} C_DIS
LIN {X 0.099,Y -568.157,Z 551.188,A 0.000,B 0.000,C 90.000,E1 69.826} C_DIS
LIN {X -0.224,Y -562.001,Z 551.185,A 0.000,B 0.000,C 90.000,E1 69.390} C_DIS
LIN {X 0.154,Y -557.333,Z 551.184,A 0.000,B 0.000,C 90.000,E1 69.028} C_DIS
LIN {X -0.075,Y -549.847,Z 551.181,A 0.000,B 0.000,C 90.000,E1 68.592} C_DIS
LIN {X -0.222,Y -543.063,Z 551.179,A 0.000,B 0.000,C 90.000,E1 68.230} C_DIS
LIN {X -0.255,Y -537.704,Z 551.178,A 0.000,B 0.000,C 90.000,E1 67.975} C_DIS
LIN {X -0.270,Y -530.672,Z 551.176,A 0.000,B 0.000,C 90.000,E1 67.667} C_DIS
LIN {X -0.251,Y -518.368,Z 551.173,A 0.000,B 0.000,C 90.000,E1 67.177} C_DIS
LIN {X -0.156,Y -509.281,Z 551.171,A 0.000,B 0.000,C 90.000,E1 66.847} C_DIS
LIN {X -0.084,Y -495.062,Z 551.169,A 0.000,B 0.000,C 90.000,E1 66.357} C_DIS
LIN {X -0.067,Y -468.851,Z 551.164,A 0.000,B 0.000,C 90.000,E1 65.485} C_DIS
LIN {X -0.172,Y -461.527,Z 551.162,A 0.000,B 0.000,C 90.000,E1 65.229} C_DIS
LIN {X -0.204,Y -461.514,Z 551.162,A 0.000,B 0.000,C 90.000,E1 65.229} C_DIS
LIN {X 0.060,Y -455.486,Z 551.144,A 0.000,B 0.000,C 90.000,E1 61.897} C_DIS
LIN {X 0.066,Y -445.536,Z 551.119,A 0.000,B 0.000,C 90.000,E1 57.375} C_DIS
LIN {X -0.118,Y -443.741,Z 551.113,A 0.000,B 0.000,C 90.000,E1 56.421} C_DIS
LIN {X -0.082,Y -440.921,Z 551.107,A 0.000,B 0.000,C 90.000,E1 55.308} C_DIS
LIN {X -0.122,Y -440.919,Z 551.107,A 0.000,B 0.000,C 90.000,E1 55.308} C_DIS
LIN {X -0.012,Y -442.841,Z 551.101,A 0.000,B 0.000,C 90.000,E1 54.116} C_DIS
LIN {X 0.067,Y -446.023,Z 551.090,A 0.000,B 0.000,C 90.000,E1 52.145} C_DIS
LIN {X 0.052,Y -447.596,Z 551.084,A 0.000,B 0.000,C 90.000,E1 51.170} C_DIS
LIN {X 0.098,Y -449.953,Z 551.075,A 0.000,B 0.000,C 90.000,E1 49.542} C_DIS
LIN {X 0.143,Y -452.244,Z 551.066,A 0.000,B 0.000,C 90.000,E1 47.919} C_DIS
LIN {X -0.114,Y -453.912,Z 551.059,A 0.000,B 0.000,C 90.000,E1 46.662} C_DIS
LIN {X 0.273,Y -454.989,Z 551.054,A 0.000,B 0.000,C 90.000,E1 45.648} C_DIS
LIN {X 0.020,Y -455.828,Z 551.048,A 0.000,B 0.000,C 90.000,E1 44.717} C_DIS
LIN {X -0.247,Y -456.375,Z 551.045,A 0.000,B 0.000,C 90.000,E1 44.109} C_DIS
LIN {X 0.199,Y -457.104,Z 551.038,A 0.000,B 0.000,C 90.000,E1 42.771} C_DIS
LIN {X 0.007,Y -457.596,Z 551.031,A 0.000,B 0.000,C 90.000,E1 41.515} C_DIS
LIN {X -0.136,Y -457.893,Z 551.024,A 0.000,B 0.000,C 90.000,E1 40.253} C_DIS
LIN {X 0.018,Y -457.876,Z 551.016,A 0.000,B 0.000,C 90.000,E1 38.955} C_DIS
LIN {X -0.034,Y -457.714,Z 551.008,A 0.000,B 0.000,C 90.000,E1 37.363} C_DIS
LIN {X -0.092,Y -457.388,Z 551.000,A 0.000,B 0.000,C 90.000,E1 36.091} C_DIS
LIN {X -0.048,Y -456.780,Z 550.992,A 0.000,B 0.000,C 90.000,E1 34.485} C_DIS
LIN {X -0.021,Y -456.140,Z 550.983,A 0.000,B 0.000,C 90.000,E1 32.880} C_DIS
LIN {X 0.123,Y -455.579,Z 550.974,A 0.000,B 0.000,C 90.000,E1 31.258} C_DIS
LIN {X 0.124,Y -454.916,Z 550.963,A 0.000,B 0.000,C 90.000,E1 29.333} C_DIS
LIN {X -0.234,Y -454.123,Z 550.951,A 0.000,B 0.000,C 90.000,E1 27.129} C_DIS
LIN {X 0.003,Y -453.364,Z 550.938,A 0.000,B 0.000,C 90.000,E1 24.847} C_DIS
LIN {X 0.141,Y -452.856,Z 550.927,A 0.000,B 0.000,C 90.000,E1 22.898} C_DIS
LIN {X -0.029,Y -452.422,Z 550.915,A 0.000,B 0.000,C 90.000,E1 20.663} C_DIS
LIN {X 0.200,Y -452.090,Z 550.901,A 0.000,B 0.000,C 90.000,E1 18.055} C_DIS
LIN {X -0.104,Y -452.130,Z 550.884,A 0.000,B 0.000,C 90.000,E1 15.190} C_DIS
LIN {X 0.044,Y -452.540,Z 550.870,A 0.000,B 0.000,C 90.000,E1 12.591} C_DIS
LIN {X -0.202,Y -453.254,Z 550.857,A 0.000,B 0.000,C 90.000,E1 10.366} C_DIS
LIN {X -0.119,Y -453.953,Z 550.849,A 0.000,B 0.000,C 90.000,E1 8.746} C_DIS
LIN {X -0.038,Y -455.219,Z 550.836,A 0.000,B 0.000,C 90.000,E1 6.486} C_DIS
LIN {X 0.200,Y -456.475,Z 550.825,A 0.000,B 0.000,C 90.000,E1 4.531} C_DIS
LIN {X -0.156,Y -459.058,Z 550.808,A 0.000,B 0.000,C 90.000,E1 1.375} C_DIS
LIN {X 0.120,Y -461.317,Z 550.795,A 0.000,B 0.000,C 90.000,E1 359.141} C_DIS
LIN {X -0.004,Y -463.617,Z 550.785,A 0.000,B 0.000,C 90.000,E1 357.249} C_DIS
LIN {X -0.047,Y -467.045,Z 550.771,A 0.000,B 0.000,C 90.000,E1 354.723} C_DIS
LIN {X 0.067,Y -469.610,Z 550.760,A 0.000,B 0.000,C 90.000,E1 352.818} C_DIS
LIN {X 0.022,Y -471.719,Z 550.751,A 0.000,B 0.000,C 90.000,E1 351.254} C_DIS
LIN {X -0.019,Y -475.365,Z 550.738,A 0.000,B 0.000,C 90.000,E1 348.757} C_DIS
LIN {X 0.217,Y -477.876,Z 550.729,A 0.000,B 0.000,C 90.000,E1 347.173} C_DIS
LIN {X -0.141,Y -481.524,Z 550.717,A 0.000,B 0.000,C 90.000,E1 345.046} C_DIS
LIN {X 0.189,Y -486.620,Z 550.701,A 0.000,B 0.000,C 90.000,E1 342.236} C_DIS
LIN {X -0.013,Y -490.200,Z 550.691,A 0.000,B 0.000,C 90.000,E1 340.423} C_DIS
LIN {X 0.024,Y -493.760,Z 550.681,A 0.000,B 0.000,C 90.000,E1 338.592} C_DIS
LIN {X 0.211,Y -496.121,Z 550.674,A 0.000,B 0.000,C 90.000,E1 337.358} C_DIS
LIN {X 0.032,Y -498.945,Z 550.666,A 0.000,B 0.000,C 90.000,E1 335.869} C_DIS
LIN {X 0.100,Y -501.665,Z 550.658,A 0.000,B 0.000,C 90.000,E1 334.357} C_DIS
LIN {X 0.062,Y -504.867,Z 550.648,A 0.000,B 0.000,C 90.000,E1 332.564} C_DIS
LIN {X 0.252,Y -507.412,Z 550.639,A 0.000,B 0.000,C 90.000,E1 331.051} C_DIS
LIN {X 0.032,Y -511.026,Z 550.628,A 0.000,B 0.000,C 90.000,E1 328.997} C_DIS
LIN {X -0.102,Y -513.613,Z 550.620,A 0.000,B 0.000,C 90.000,E1 327.533} C_DIS
LIN {X 0.005,Y -516.783,Z 550.610,A 0.000,B 0.000,C 90.000,E1 325.754} C_DIS
LIN {X 0.107,Y -519.396,Z 550.602,A 0.000,B 0.000,C 90.000,E1 324.276} C_DIS
LIN {X -0.207,Y -522.494,Z 550.592,A 0.000,B 0.000,C 90.000,E1 322.557} C_DIS
LIN {X -0.170,Y -526.351,Z 550.581,A 0.000,B 0.000,C 90.000,E1 320.517} C_DIS
LIN {X -0.226,Y -532.473,Z 550.565,A 0.000,B 0.000,C 90.000,E1 317.634} C_DIS
LIN {X 0.325,Y -537.156,Z 550.553,A 0.000,B 0.000,C 90.000,E1 315.567} C_DIS
LIN {X -0.139,Y -542.887,Z 550.541,A 0.000,B 0.000,C 90.000,E1 313.338} C_DIS
LIN {X -0.105,Y -546.504,Z 550.533,A 0.000,B 0.000,C 90.000,E1 311.919} C_DIS
LIN {X -0.009,Y -549.273,Z 550.527,A 0.000,B 0.000,C 90.000,E1 310.782} C_DIS
LIN {X 0.024,Y -550.817,Z 550.523,A 0.000,B 0.000,C 90.000,E1 310.216} C_DIS
LIN {X 0.075,Y -551.512,Z 550.522,A 0.000,B 0.000,C 90.000,E1 309.930} C_DIS
LIN {X 0.192,Y -553.496,Z 550.519,A 0.000,B 0.000,C 90.000,E1 309.358} C_DIS
LIN {X -0.030,Y -553.894,Z 550.518,A 0.000,B 0.000,C 90.000,E1 309.241} C_DIS
LIN {X -0.002,Y -556.556,Z 550.515,A 0.000,B 0.000,C 90.000,E1 308.749} C_DIS
LIN {X 0.182,Y -559.032,Z 550.513,A 0.000,B 0.000,C 90.000,E1 308.382} C_DIS
LIN {X 0.269,Y -561.569,Z 550.512,A 0.000,B 0.000,C 90.000,E1 308.096} C_DIS
LIN {X 0.158,Y -562.679,Z 550.511,A 0.000,B 0.000,C 90.000,E1 307.971} C_DIS
LIN {X 0.041,Y -565.934,Z 550.509,A 0.000,B 0.000,C 90.000,E1 307.684} C_DIS
LIN {X -0.051,Y -567.063,Z 550.509,A 0.000,B 0.000,C 90.000,E1 307.569} C_DIS
LIN {X -0.040,Y -568.403,Z 550.508,A 0.000,B 0.000,C 90.000,E1 307.443} C_DIS
LIN {X -0.105,Y -577.643,Z 550.504,A 0.000,B 0.000,C 90.000,E1 306.710} C_DIS
LIN {X -0.058,Y -581.690,Z 550.502,A 0.000,B 0.000,C 90.000,E1 306.377} C_DIS
LIN {X -0.174,Y -586.857,Z 550.500,A 0.000,B 0.000,C 90.000,E1 305.931} C_DIS
LIN {X -0.074,Y -591.913,Z 550.497,A 0.000,B 0.000,C 90.000,E1 305.438} C_DIS
LIN {X 0.263,Y -595.704,Z 550.495,A 0.000,B 0.000,C 90.000,E1 305.025} C_DIS
LIN {X -0.088,Y -602.976,Z 550.490,A 0.000,B 0.000,C 90.000,E1 304.278} C_DIS
LIN {X -0.162,Y -611.330,Z 550.485,A 0.000,B 0.000,C 90.000,E1 303.372} C_DIS
LIN {X -0.103,Y -620.477,Z 550.480,A 0.000,B 0.000,C 90.000,E1 302.339} C_DIS
LIN {X 0.193,Y -624.921,Z 550.477,A 0.000,B 0.000,C 90.000,E1 301.799} C_DIS
LIN {X -0.341,Y -629.061,Z 550.474,A 0.000,B 0.000,C 90.000,E1 301.337} C_DIS
LIN {X 0.017,Y -632.896,Z 550.471,A 0.000,B 0.000,C 90.000,E1 300.797} C_DIS
LIN {X 0.081,Y -636.356,Z 550.468,A 0.000,B 0.000,C 90.000,E1 300.285} C_DIS
LIN {X -0.036,Y -640.040,Z 550.465,A 0.000,B 0.000,C 90.000,E1 299.667} C_DIS
LIN {X 0.112,Y -642.933,Z 550.461,A 0.000,B 0.000,C 90.000,E1 299.027} C_DIS
LIN {X 0.067,Y -645.657,Z 550.457,A 0.000,B 0.000,C 90.000,E1 298.281} C_DIS
LIN {X 0.000,Y -650.927,Z 550.449,A 0.000,B 0.000,C 90.000,E1 296.796} C_DIS
LIN {X 0.095,Y -651.691,Z 550.448,A 0.000,B 0.000,C 90.000,E1 296.539} C_DIS
LIN {X 0.008,Y -652.647,Z 550.445,A 0.000,B 0.000,C 90.000,E1 296.052} C_DIS
LIN {X 0.113,Y -652.913,Z 550.443,A 0.000,B 0.000,C 90.000,E1 295.796} C_DIS
LIN {X -0.264,Y -652.201,Z 550.441,A 0.000,B 0.000,C 90.000,E1 295.335} C_DIS
LIN {X -0.160,Y -651.376,Z 550.439,A 0.000,B 0.000,C 90.000,E1 295.079} C_DIS
LIN {X -0.010,Y -649.514,Z 550.437,A 0.000,B 0.000,C 90.000,E1 294.695} C_DIS
LIN {X -0.230,Y -648.572,Z 550.437,A 0.000,B 0.000,C 90.000,E1 294.591} C_DIS
LIN {X -0.184,Y -647.407,Z 550.436,A 0.000,B 0.000,C 90.000,E1 294.463} C_DIS
LIN {X -0.137,Y -645.510,Z 550.435,A 0.000,B 0.000,C 90.000,E1 294.335} C_DIS
LIN {X 0.171,Y -644.403,Z 550.435,A 0.000,B 0.000,C 90.000,E1 294.259} C_DIS
LIN {X -0.025,Y -642.667,Z 550.434,A 0.000,B 0.000,C 90.000,E1 294.131} C_DIS
LIN {X -0.160,Y -641.350,Z 550.433,A 0.000,B 0.000,C 90.000,E1 294.027} C_DIS
LIN {X -0.032,Y -639.381,Z 550.433,A 0.000,B 0.000,C 90.000,E1 293.898} C_DIS
LIN {X -0.175,Y -632.589,Z 550.431,A 0.000,B 0.000,C 90.000,E1 293.567} C_DIS
LIN {X 0.107,Y -624.879,Z 550.429,A 0.000,B 0.000,C 90.000,E1 293.259} C_DIS
LIN {X -0.267,Y -619.358,Z 550.428,A 0.000,B 0.000,C 90.000,E1 293.078} C_DIS
LIN {X -0.013,Y -609.596,Z 550.426,A 0.000,B 0.000,C 90.000,E1 292.717} C_DIS
LIN {X -0.223,Y -595.614,Z 550.424,A 0.000,B 0.000,C 90.000,E1 292.280} C_DIS
LIN {X 0.276,Y -585.574,Z 550.422,A 0.000,B 0.000,C 90.000,E1 291.897} C_DIS
LIN {X -0.213,Y -580.764,Z 550.421,A 0.000,B 0.000,C 90.000,E1 291.770} C_DIS
LIN {X 0.017,Y -576.284,Z 550.420,A 0.000,B 0.000,C 90.000,E1 291.535} C_DIS
LIN {X -0.137,Y -573.598,Z 550.419,A 0.000,B 0.000,C 90.000,E1 291.408} C_DIS
LIN {X 0.057,Y -570.783,Z 550.418,A 0.000,B 0.000,C 90.000,E1 291.173} C_DIS
LIN {X 0.093,Y -569.545,Z 550.417,A 0.000,B 0.000,C 90.000,E1 290.972} C_DIS
LIN {X 0.051,Y -569.524,Z 550.417,A 0.000,B 0.000,C 90.000,E1 290.972} C_DIS
LIN {X -0.022,Y -569.031,Z 550.414,A 0.000,B 0.000,C 90.000,E1 290.556} C_DIS
LIN {X 0.163,Y -568.994,Z 550.405,A 0.000,B 0.000,C 90.000,E1 288.906} C_DIS
LIN {X -0.291,Y -568.776,Z 550.398,A 0.000,B 0.000,C 90.000,E1 287.583} C_DIS
LIN {X 0.170,Y -568.464,Z 550.391,A 0.000,B 0.000,C 90.000,E1 286.441} C_DIS
LIN {X 0.243,Y -567.855,Z 550.384,A 0.000,B 0.000,C 90.000,E1 285.064} C_DIS
LIN {X -0.162,Y -567.226,Z 550.378,A 0.000,B 0.000,C 90.000,E1 284.008} C_DIS
LIN {X 0.287,Y -566.433,Z 550.370,A 0.000,B 0.000,C 90.000,E1 282.591} C_DIS
LIN {X 0.209,Y -565.560,Z 550.361,A 0.000,B 0.000,C 90.000,E1 280.950} C_DIS
LIN {X 0.243,Y -564.435,Z 550.349,A 0.000,B 0.000,C 90.000,E1 278.746} C_DIS
LIN {X 0.089,Y -563.561,Z 550.338,A 0.000,B 0.000,C 90.000,E1 276.834} C_DIS
LIN {X 0.009,Y -563.110,Z 550.332,A 0.000,B 0.000,C 90.000,E1 275.739} C_DIS
LIN {X -0.080,Y -562.678,Z 550.326,A 0.000,B 0.000,C 90.000,E1 274.645} C_DIS
LIN {X -0.121,Y -562.106,Z 550.318,A 0.000,B 0.000,C 90.000,E1 273.269} C_DIS
LIN {X -0.049,Y -561.309,Z 550.309,A 0.000,B 0.000,C 90.000,E1 271.604} C_DIS
LIN {X -0.223,Y -560.724,Z 550.303,A 0.000,B 0.000,C 90.000,E1 270.516} C_DIS
LIN {X -0.125,Y -559.578,Z 550.292,A 0.000,B 0.000,C 90.000,E1 268.568} C_DIS
LIN {X 0.163,Y -559.106,Z 550.287,A 0.000,B 0.000,C 90.000,E1 267.707} C_DIS
LIN {X 0.142,Y -558.083,Z 550.278,A 0.000,B 0.000,C 90.000,E1 266.045} C_DIS
LIN {X 0.052,Y -557.229,Z 550.270,A 0.000,B 0.000,C 90.000,E1 264.666} C_DIS
LIN {X 0.066,Y -556.102,Z 550.261,A 0.000,B 0.000,C 90.000,E1 262.996} C_DIS
LIN {X 0.076,Y -555.027,Z 550.253,A 0.000,B 0.000,C 90.000,E1 261.602} C_DIS
LIN {X -0.176,Y -554.203,Z 550.249,A 0.000,B 0.000,C 90.000,E1 260.792} C_DIS
LIN {X -0.194,Y -552.455,Z 550.241,A 0.000,B 0.000,C 90.000,E1 259.398} C_DIS
LIN {X -0.141,Y -550.848,Z 550.233,A 0.000,B 0.000,C 90.000,E1 257.993} C_DIS
LIN {X -0.120,Y -549.232,Z 550.225,A 0.000,B 0.000,C 90.000,E1 256.589} C_DIS
LIN {X 0.231,Y -547.048,Z 550.216,A 0.000,B 0.000,C 90.000,E1 254.866} C_DIS
LIN {X 0.215,Y -545.410,Z 550.210,A 0.000,B 0.000,C 90.000,E1 253.740} C_DIS
LIN {X -0.118,Y -543.116,Z 550.202,A 0.000,B 0.000,C 90.000,E1 252.362} C_DIS
LIN {X 0.190,Y -540.749,Z 550.194,A 0.000,B 0.000,C 90.000,E1 250.913} C_DIS
LIN {X -0.097,Y -538.695,Z 550.188,A 0.000,B 0.000,C 90.000,E1 249.806} C_DIS
LIN {X -0.171,Y -535.202,Z 550.178,A 0.000,B 0.000,C 90.000,E1 248.103} C_DIS
LIN {X 0.160,Y -532.771,Z 550.172,A 0.000,B 0.000,C 90.000,E1 246.922} C_DIS
LIN {X 0.155,Y -529.476,Z 550.164,A 0.000,B 0.000,C 90.000,E1 245.485} C_DIS
LIN {X 0.138,Y -526.681,Z 550.158,A 0.000,B 0.000,C 90.000,E1 244.332} C_DIS
LIN {X 0.088,Y -523.697,Z 550.151,A 0.000,B 0.000,C 90.000,E1 243.179} C_DIS
LIN {X 0.049,Y -519.053,Z 550.141,A 0.000,B 0.000,C 90.000,E1 241.435} C_DIS
LIN {X -0.212,Y -515.084,Z 550.133,A 0.000,B 0.000,C 90.000,E1 239.999} C_DIS
LIN {X 0.156,Y -512.547,Z 550.128,A 0.000,B 0.000,C 90.000,E1 239.076} C_DIS
LIN {X -0.080,Y -507.161,Z 550.118,A 0.000,B 0.000,C 90.000,E1 237.327} C_DIS
LIN {X 0.122,Y -501.861,Z 550.109,A 0.000,B 0.000,C 90.000,E1 235.515} C_DIS
LIN {X -0.066,Y -497.605,Z 550.100,A 0.000,B 0.000,C 90.000,E1 234.036} C_DIS
LIN {X 0.068,Y -491.810,Z 550.088,A 0.000,B 0.000,C 90.000,E1 231.904} C_DIS
LIN {X 0.090,Y -485.334,Z 550.075,A 0.000,B 0.000,C 90.000,E1 229.461} C_DIS
LIN {X -0.064,Y -480.573,Z 550.065,A 0.000,B 0.000,C 90.000,E1 227.634} C_DIS
LIN {X -0.239,Y -475.160,Z 550.053,A 0.000,B 0.000,C 90.000,E1 225.486} C_DIS
LIN {X 0.029,Y -470.660,Z 550.042,A 0.000,B 0.000,C 90.000,E1 223.581} C_DIS
LIN {X 0.189,Y -466.264,Z 550.032,A 0.000,B 0.000,C 90.000,E1 221.676} C_DIS
LIN {X 0.222,Y -462.663,Z 550.023,A 0.000,B 0.000,C 90.000,E1 220.092} C_DIS
LIN {X -0.081,Y -458.457,Z 550.012,A 0.000,B 0.000,C 90.000,E1 218.222} C_DIS
LIN {X -0.042,Y -454.293,Z 550.002,A 0.000,B 0.000,C 90.000,E1 216.297} C_DIS
LIN {X -0.023,Y -449.605,Z 549.989,A 0.000,B 0.000,C 90.000,E1 214.040} C_DIS
LIN {X 0.051,Y -445.725,Z 549.978,A 0.000,B 0.000,C 90.000,E1 212.084} C_DIS
LIN {X 0.138,Y -440.766,Z 549.964,A 0.000,B 0.000,C 90.000,E1 209.461} C_DIS
LIN {X -0.080,Y -437.823,Z 549.955,A 0.000,B 0.000,C 90.000,E1 207.847} C_DIS
LIN {X 0.056,Y -434.479,Z 549.944,A 0.000,B 0.000,C 90.000,E1 205.848} C_DIS
LIN {X -0.088,Y -431.243,Z 549.933,A 0.000,B 0.000,C 90.000,E1 203.875} C_DIS
LIN {X 0.136,Y -428.160,Z 549.922,A 0.000,B 0.000,C 90.000,E1 201.844} C_DIS
LIN {X -0.073,Y -423.987,Z 549.905,A 0.000,B 0.000,C 90.000,E1 198.852} C_DIS
LIN {X 0.050,Y -420.481,Z 549.890,A 0.000,B 0.000,C 90.000,E1 196.134} C_DIS
LIN {X -0.049,Y -417.698,Z 549.877,A 0.000,B 0.000,C 90.000,E1 193.772} C_DIS
LIN {X -0.055,Y -415.858,Z 549.869,A 0.000,B 0.000,C 90.000,E1 192.411} C_DIS
LIN {X -0.060,Y -412.767,Z 549.856,A 0.000,B 0.000,C 90.000,E1 190.018} C_DIS
LIN {X 0.152,Y -409.695,Z 549.840,A 0.000,B 0.000,C 90.000,E1 187.239} C_DIS
LIN {X 0.159,Y -407.335,Z 549.827,A 0.000,B 0.000,C 90.000,E1 184.821} C_DIS
LIN {X 0.041,Y -404.833,Z 549.812,A 0.000,B 0.000,C 90.000,E1 182.064} C_DIS
LIN {X -0.125,Y -403.194,Z 549.800,A 0.000,B 0.000,C 90.000,E1 180.000} C_DIS
LIN {X 0.037,Y -401.800,Z 549.786,A 0.000,B 0.000,C 90.000,E1 177.535} C_DIS
LIN {X 0.200,Y -400.818,Z 549.773,A 0.000,B 0.000,C 90.000,E1 175.065} C_DIS
LIN {X -0.016,Y -400.312,Z 549.761,A 0.000,B 0.000,C 90.000,E1 172.996} C_DIS
LIN {X -0.082,Y -400.127,Z 549.751,A 0.000,B 0.000,C 90.000,E1 171.254} C_DIS
LIN {X -0.140,Y -400.129,Z 549.742,A 0.000,B 0.000,C 90.000,E1 169.511} C_DIS
LIN {X -0.087,Y -400.408,Z 549.726,A 0.000,B 0.000,C 90.000,E1 166.700} C_DIS
LIN {X 0.152,Y -401.160,Z 549.711,A 0.000,B 0.000,C 90.000,E1 163.866} C_DIS
LIN {X -0.023,Y -402.171,Z 549.695,A 0.000,B 0.000,C 90.000,E1 161.094} C_DIS
LIN {X -0.223,Y -403.204,Z 549.683,A 0.000,B 0.000,C 90.000,E1 159.028} C_DIS
LIN {X 0.142,Y -404.581,Z 549.670,A 0.000,B 0.000,C 90.000,E1 156.538} C_DIS
LIN {X 0.086,Y -405.864,Z 549.658,A 0.000,B 0.000,C 90.000,E1 154.460} C_DIS
LIN {X -0.037,Y -406.970,Z 549.649,A 0.000,B 0.000,C 90.000,E1 152.743} C_DIS
LIN {X 0.039,Y -407.994,Z 549.639,A 0.000,B 0.000,C 90.000,E1 151.001} C_DIS
LIN {X -0.029,Y -408.958,Z 549.629,A 0.000,B 0.000,C 90.000,E1 149.282} C_DIS
LIN {X 0.053,Y -409.842,Z 549.618,A 0.000,B 0.000,C 90.000,E1 147.199} C_DIS
LIN {X 0.027,Y -410.544,Z 549.606,A 0.000,B 0.000,C 90.000,E1 145.135} C_DIS
LIN {X 0.001,Y -410.951,Z 549.597,A 0.000,B 0.000,C 90.000,E1 143.417} C_DIS
LIN {X -0.014,Y -411.264,Z 549.587,A 0.000,B 0.000,C 90.000,E1 141.698} C_DIS
LIN {X -0.256,Y -411.384,Z 549.580,A 0.000,B 0.000,C 90.000,E1 140.356} C_DIS
LIN {X -0.062,Y -411.461,Z 549.570,A 0.000,B 0.000,C 90.000,E1 138.609} C_DIS
LIN {X -0.016,Y -411.519,Z 549.559,A 0.000,B 0.000,C 90.000,E1 136.539} C_DIS
LIN {X 0.157,Y -411.708,Z 549.545,A 0.000,B 0.000,C 90.000,E1 134.109} C_DIS
LIN {X -0.093,Y -411.834,Z 549.534,A 0.000,B 0.000,C 90.000,E1 132.081} C_DIS
LIN {X -0.054,Y -411.757,Z 549.526,A 0.000,B 0.000,C 90.000,E1 130.701} C_DIS
LIN {X 0.129,Y -411.634,Z 549.520,A 0.000,B 0.000,C 90.000,E1 129.644} C_DIS
LIN {X 0.048,Y -411.316,Z 549.515,A 0.000,B 0.000,C 90.000,E1 128.624} C_DIS
LIN {X -0.053,Y -410.807,Z 549.509,A 0.000,B 0.000,C 90.000,E1 127.569} C_DIS
LIN {X -0.092,Y -410.810,Z 549.509,A 0.000,B 0.000,C 90.000,E1 127.569} C_DIS
LIN {X -0.023,Y -415.769,Z 549.499,A 0.000,B 0.000,C 90.000,E1 125.884} C_DIS
LIN {X 0.083,Y -425.215,Z 549.479,A 0.000,B 0.000,C 90.000,E1 122.133} C_DIS
LIN {X 0.017,Y -430.216,Z 549.469,A 0.000,B 0.000,C 90.000,E1 120.463} C_DIS
LIN {X 0.016,Y -431.128,Z 549.467,A 0.000,B 0.000,C 90.000,E1 120.129} C_DIS
LIN {X -0.038,Y -440.232,Z 549.447,A 0.000,B 0.000,C 90.000,E1 116.488} C_DIS
LIN {X 0.188,Y -443.486,Z 549.441,A 0.000,B 0.000,C 90.000,E1 115.335} C_DIS
LIN {X 0.148,Y -443.524,Z 549.441,A 0.000,B 0.000,C 90.000,E1 115.335} C_DIS
LIN {X -0.102,Y -463.264,Z 549.436,A 0.000,B 0.000,C 90.000,E1 114.515} C_DIS
LIN {X -0.050,Y -482.412,Z 549.432,A 0.000,B 0.000,C 90.000,E1 113.695} C_DIS
LIN {X 0.024,Y -496.071,Z 549.428,A 0.000,B 0.000,C 90.000,E1 113.078} C_DIS
LIN {X 0.154,Y -505.971,Z 549.426,A 0.000,B 0.000,C 90.000,E1 112.589} C_DIS
LIN {X 0.115,Y -516.168,Z 549.423,A 0.000,B 0.000,C 90.000,E1 112.099} C_DIS
LIN {X 0.080,Y -522.625,Z 549.421,A 0.000,B 0.000,C 90.000,E1 111.770} C_DIS
LIN {X 0.054,Y -534.056,Z 549.418,A 0.000,B 0.000,C 90.000,E1 111.153} C_DIS
LIN {X 0.149,Y -541.973,Z 549.415,A 0.000,B 0.000,C 90.000,E1 110.684} C_DIS
LIN {X 0.059,Y -548.083,Z 549.413,A 0.000,B 0.000,C 90.000,E1 110.301} C_DIS
LIN {X 0.083,Y -554.008,Z 549.411,A 0.000,B 0.000,C 90.000,E1 109.885} C_DIS
LIN {X -0.010,Y -559.630,Z 549.408,A 0.000,B 0.000,C 90.000,E1 109.450} C_DIS
LIN {X 0.145,Y -565.085,Z 549.405,A 0.000,B 0.000,C 90.000,E1 108.960} C_DIS
LIN {X -0.197,Y -570.249,Z 549.403,A 0.000,B 0.000,C 90.000,E1 108.489} C_DIS
LIN {X -0.050,Y -575.119,Z 549.400,A 0.000,B 0.000,C 90.000,E1 107.946} C_DIS
LIN {X 0.207,Y -581.158,Z 549.396,A 0.000,B 0.000,C 90.000,E1 107.166} C_DIS
LIN {X -0.016,Y -585.733,Z 549.392,A 0.000,B 0.000,C 90.000,E1 106.551} C_DIS
LIN {X -0.188,Y -590.300,Z 549.388,A 0.000,B 0.000,C 90.000,E1 105.898} C_DIS
LIN {X -0.115,Y -594.414,Z 549.385,A 0.000,B 0.000,C 90.000,E1 105.245} C_DIS
LIN {X 0.083,Y -596.691,Z 549.382,A 0.000,B 0.000,C 90.000,E1 104.828} C_DIS
LIN {X 0.147,Y -599.011,Z 549.380,A 0.000,B 0.000,C 90.000,E1 104.426} C_DIS
LIN {X 0.152,Y -605.397,Z 549.374,A 0.000,B 0.000,C 90.000,E1 103.244} C_DIS
LIN {X -0.305,Y -610.905,Z 549.368,A 0.000,B 0.000,C 90.000,E1 102.243} C_DIS
LIN {X 0.331,Y -614.136,Z 549.364,A 0.000,B 0.000,C 90.000,E1 101.535} C_DIS
LIN {X -0.096,Y -615.980,Z 549.362,A 0.000,B 0.000,C 90.000,E1 101.186} C_DIS
LIN {X -0.207,Y -619.285,Z 549.358,A 0.000,B 0.000,C 90.000,E1 100.423} C_DIS
LIN {X -0.341,Y -624.480,Z 549.351,A 0.000,B 0.000,C 90.000,E1 99.151} C_DIS
LIN {X 0.337,Y -629.797,Z 549.344,A 0.000,B 0.000,C 90.000,E1 97.814} C_DIS
LIN {X -0.035,Y -633.847,Z 549.338,A 0.000,B 0.000,C 90.000,E1 96.834} C_DIS
LIN {X 0.278,Y -637.819,Z 549.332,A 0.000,B 0.000,C 90.000,E1 95.796} C_DIS
LIN {X -0.052,Y -641.242,Z 549.327,A 0.000,B 0.000,C 90.000,E1 94.821} C_DIS
LIN {X -0.091,Y -643.566,Z 549.323,A 0.000,B 0.000,C 90.000,E1 94.073} C_DIS
LIN {X -0.304,Y -646.321,Z 549.317,A 0.000,B 0.000,C 90.000,E1 93.094} C_DIS
LIN {X -0.111,Y -647.526,Z 549.314,A 0.000,B 0.000,C 90.000,E1 92.579} C_DIS
LIN {X -0.122,Y -649.055,Z 549.310,A 0.000,B 0.000,C 90.000,E1 91.835} C_DIS
LIN {X -0.098,Y -650.221,Z 549.306,A 0.000,B 0.000,C 90.000,E1 91.088} C_DIS
LIN {X -0.079,Y -651.100,Z 549.302,A 0.000,B 0.000,C 90.000,E1 90.344} C_DIS
LIN {X -0.050,Y -651.717,Z 549.298,A 0.000,B 0.000,C 90.000,E1 89.599} C_DIS
LIN {X -0.223,Y -651.906,Z 549.292,A 0.000,B 0.000,C 90.000,E1 88.625} C_DIS
LIN {X -0.169,Y -651.714,Z 549.288,A 0.000,B 0.000,C 90.000,E1 87.879} C_DIS
LIN {X 0.068,Y -651.418,Z 549.285,A 0.000,B 0.000,C 90.000,E1 87.364} C_DIS
LIN {X -0.090,Y -650.460,Z 549.280,A 0.000,B 0.000,C 90.000,E1 86.388} C_DIS
LIN {X -0.041,Y -649.485,Z 549.276,A 0.000,B 0.000,C 90.000,E1 85.641} C_DIS
LIN {X -0.228,Y -647.821,Z 549.270,A 0.000,B 0.000,C 90.000,E1 84.666} C_DIS
LIN {X -0.144,Y -646.351,Z 549.266,A 0.000,B 0.000,C 90.000,E1 83.913} C_DIS
LIN {X 0.099,Y -645.207,Z 549.263,A 0.000,B 0.000,C 90.000,E1 83.394} C_DIS
LIN {X 0.087,Y -643.221,Z 549.259,A 0.000,B 0.000,C 90.000,E1 82.648} C_DIS
LIN {X -0.035,Y -640.269,Z 549.254,A 0.000,B 0.000,C 90.000,E1 81.659} C_DIS
LIN {X -0.287,Y -636.972,Z 549.248,A 0.000,B 0.000,C 90.000,E1 80.679} C_DIS
LIN {X -0.192,Y -634.274,Z 549.244,A 0.000,B 0.000,C 90.000,E1 79.916} C_DIS
LIN {X -0.231,Y -631.371,Z 549.240,A 0.000,B 0.000,C 90.000,E1 79.162} C_DIS
LIN {X -0.306,Y -628.188,Z 549.235,A 0.000,B 0.000,C 90.000,E1 78.409} C_DIS
LIN {X -0.290,Y -624.775,Z 549.231,A 0.000,B 0.000,C 90.000,E1 77.645} C_DIS
LIN {X -0.305,Y -621.174,Z 549.227,A 0.000,B 0.000,C 90.000,E1 76.881} C_DIS
LIN {X -0.136,Y -618.622,Z 549.224,A 0.000,B 0.000,C 90.000,E1 76.353} C_DIS
LIN {X -0.032,Y -615.048,Z 549.221,A 0.000,B 0.000,C 90.000,E1 75.700} C_DIS
LIN {X 0.088,Y -612.170,Z 549.218,A 0.000,B 0.000,C 90.000,E1 75.172} C_DIS
LIN {X 0.091,Y -607.393,Z 549.213,A 0.000,B 0.000,C 90.000,E1 74.393} C_DIS
LIN {X 0.050,Y -602.145,Z 549.209,A 0.000,B 0.000,C 90.000,E1 73.614} C_DIS
LIN {X 0.071,Y -598.328,Z 549.206,A 0.000,B 0.000,C 90.000,E1 73.087} C_DIS
LIN {X 0.175,Y -592.932,Z 549.202,A 0.000,B 0.000,C 90.000,E1 72.417} C_DIS
LIN {X 0.122,Y -588.262,Z 549.200,A 0.000,B 0.000,C 90.000,E1 71.891} C_DIS
LIN {X -0.257,Y -583.116,Z 549.197,A 0.000,B 0.000,C 90.000,E1 71.402} C_DIS
LIN {X 0.009,Y -577.761,Z 549.194,A 0.000,B 0.000,C 90.000,E1 70.859} C_DIS
LIN {X -0.108,Y -572.176,Z 549.191,A 0.000,B 0.000,C 90.000,E1 70.369} C_DIS
LIN {X -0.088,Y -567.888,Z 549.189,A 0.000,B 0.000,C 90.000,E1 70.007} C_DIS
LIN {X -0.269,Y -561.839,Z 549.186,A 0.000,B 0.000,C 90.000,E1 69.571} C_DIS
LIN {X -0.121,Y -555.488,Z 549.184,A 0.000,B 0.000,C 90.000,E1 69.135} C_DIS
LIN {X 0.160,Y -548.843,Z 549.182,A 0.000,B 0.000,C 90.000,E1 68.720} C_DIS
LIN {X -0.044,Y -543.814,Z 549.180,A 0.000,B 0.000,C 90.000,E1 68.465} C_DIS
LIN {X -0.262,Y -538.522,Z 549.179,A 0.000,B 0.000,C 90.000,E1 68.230} C_DIS
LIN {X -0.056,Y -531.452,Z 549.177,A 0.000,B 0.000,C 90.000,E1 67.901} C_DIS
LIN {X -0.080,Y -520.782,Z 549.175,A 0.000,B 0.000,C 90.000,E1 67.486} C_DIS
LIN {X -0.153,Y -513.595,Z 549.173,A 0.000,B 0.000,C 90.000,E1 67.230} C_DIS
LIN {X 0.057,Y -497.419,Z 549.170,A 0.000,B 0.000,C 90.000,E1 66.666} C_DIS
LIN {X -0.219,Y -469.322,Z 549.165,A 0.000,B 0.000,C 90.000,E1 65.793} C_DIS
LIN {X -0.190,Y -462.238,Z 549.164,A 0.000,B 0.000,C 90.000,E1 65.537} C_DIS
LIN {X 0.198,Y -462.160,Z 549.164,A 0.000,B 0.000,C 90.000,E1 65.485} C_DIS
LIN {X -0.128,Y -455.440,Z 549.144,A 0.000,B 0.000,C 90.000,E1 61.897} C_DIS
LIN {X 0.187,Y -446.101,Z 549.121,A 0.000,B 0.000,C 90.000,E1 57.661} C_DIS
LIN {X 0.065,Y -443.678,Z 549.113,A 0.000,B 0.000,C 90.000,E1 56.373} C_DIS
LIN {X -0.236,Y -441.265,Z 549.108,A 0.000,B 0.000,C 90.000,E1 55.468} C_DIS
LIN {X -0.024,Y -441.266,Z 549.108,A 0.000,B 0.000,C 90.000,E1 55.435} C_DIS
LIN {X 0.164,Y -443.577,Z 549.101,A 0.000,B 0.000,C 90.000,E1 54.069} C_DIS
LIN {X -0.147,Y -446.291,Z 549.091,A 0.000,B 0.000,C 90.000,E1 52.477} C_DIS
LIN {X -0.105,Y -448.441,Z 549.084,A 0.000,B 0.000,C 90.000,E1 51.170} C_DIS
LIN {X 0.253,Y -450.389,Z 549.077,A 0.000,B 0.000,C 90.000,E1 49.828} C_DIS
LIN {X 0.009,Y -452.726,Z 549.068,A 0.000,B 0.000,C 90.000,E1 48.243} C_DIS
LIN {X 0.088,Y -454.461,Z 549.061,A 0.000,B 0.000,C 90.000,E1 46.944} C_DIS
LIN {X 0.149,Y -455.569,Z 549.056,A 0.000,B 0.000,C 90.000,E1 45.972} C_DIS
LIN {X 0.227,Y -456.468,Z 549.050,A 0.000,B 0.000,C 90.000,E1 45.000} C_DIS
LIN {X -0.013,Y -457.211,Z 549.045,A 0.000,B 0.000,C 90.000,E1 44.069} C_DIS
LIN {X 0.097,Y -457.805,Z 549.040,A 0.000,B 0.000,C 90.000,E1 43.095} C_DIS
LIN {X -0.082,Y -458.319,Z 549.032,A 0.000,B 0.000,C 90.000,E1 41.838} C_DIS
LIN {X 0.086,Y -458.637,Z 549.025,A 0.000,B 0.000,C 90.000,E1 40.539} C_DIS
LIN {X -0.015,Y -458.643,Z 549.016,A 0.000,B 0.000,C 90.000,E1 38.955} C_DIS
LIN {X -0.067,Y -458.493,Z 549.009,A 0.000,B 0.000,C 90.000,E1 37.684} C_DIS
LIN {X -0.100,Y -458.066,Z 549.000,A 0.000,B 0.000,C 90.000,E1 36.091} C_DIS
LIN {X -0.311,Y -457.324,Z 548.990,A 0.000,B 0.000,C 90.000,E1 34.199} C_DIS
LIN {X -0.061,Y -456.455,Z 548.977,A 0.000,B 0.000,C 90.000,E1 31.926} C_DIS
LIN {X 0.065,Y -455.626,Z 548.965,A 0.000,B 0.000,C 90.000,E1 29.667} C_DIS
LIN {X -0.061,Y -454.770,Z 548.952,A 0.000,B 0.000,C 90.000,E1 27.436} C_DIS
LIN {X -0.119,Y -454.044,Z 548.942,A 0.000,B 0.000,C 90.000,E1 25.515} C_DIS
LIN {X -0.084,Y -453.383,Z 548.929,A 0.000,B 0.000,C 90.000,E1 23.259} C_DIS
LIN {X 0.067,Y -452.806,Z 548.915,A 0.000,B 0.000,C 90.000,E1 20.663} C_DIS
LIN {X -0.007,Y -452.459,Z 548.902,A 0.000,B 0.000,C 90.000,E1 18.417} C_DIS
LIN {X -0.051,Y -452.397,Z 548.888,A 0.000,B 0.000,C 90.000,E1 15.843} C_DIS
LIN {X 0.173,Y -452.813,Z 548.870,A 0.000,B 0.000,C 90.000,E1 12.591} C_DIS
LIN {X -0.094,Y -453.779,Z 548.854,A 0.000,B 0.000,C 90.000,E1 9.726} C_DIS
LIN {X -0.106,Y -455.201,Z 548.838,A 0.000,B 0.000,C 90.000,E1 6.834} C_DIS
LIN {X -0.105,Y -456.642,Z 548.825,A 0.000,B 0.000,C 90.000,E1 4.588} C_DIS
LIN {X 0.001,Y -459.183,Z 548.808,A 0.000,B 0.000,C 90.000,E1 1.375} C_DIS
LIN {X 0.122,Y -461.443,Z 548.795,A 0.000,B 0.000,C 90.000,E1 359.141} C_DIS
LIN {X 0.000,Y -463.732,Z 548.785,A 0.000,B 0.000,C 90.000,E1 357.249} C_DIS
LIN {X -0.040,Y -467.131,Z 548.771,A 0.000,B 0.000,C 90.000,E1 354.723} C_DIS
LIN {X 0.076,Y -469.672,Z 548.760,A 0.000,B 0.000,C 90.000,E1 352.818} C_DIS
LIN {X 0.032,Y -471.780,Z 548.751,A 0.000,B 0.000,C 90.000,E1 351.254} C_DIS
LIN {X -0.007,Y -475.418,Z 548.738,A 0.000,B 0.000,C 90.000,E1 348.757} C_DIS
LIN {X 0.074,Y -478.428,Z 548.727,A 0.000,B 0.000,C 90.000,E1 346.881} C_DIS
LIN {X -0.127,Y -481.589,Z 548.717,A 0.000,B 0.000,C 90.000,E1 345.046} C_DIS
LIN {X 0.205,Y -486.687,Z 548.701,A 0.000,B 0.000,C 90.000,E1 342.236} C_DIS
LIN {X 0.005,Y -490.275,Z 548.691,A 0.000,B 0.000,C 90.000,E1 340.423} C_DIS
LIN {X 0.045,Y -493.834,Z 548.681,A 0.000,B 0.000,C 90.000,E1 338.592} C_DIS
LIN {X 0.182,Y -495.641,Z 548.676,A 0.000,B 0.000,C 90.000,E1 337.667} C_DIS
LIN {X -0.005,Y -498.486,Z 548.668,A 0.000,B 0.000,C 90.000,E1 336.177} C_DIS
LIN {X 0.060,Y -501.228,Z 548.659,A 0.000,B 0.000,C 90.000,E1 334.665} C_DIS
LIN {X 0.018,Y -504.454,Z 548.649,A 0.000,B 0.000,C 90.000,E1 332.871} C_DIS
LIN {X -0.111,Y -506.562,Z 548.643,A 0.000,B 0.000,C 90.000,E1 331.691} C_DIS
LIN {X 0.201,Y -509.624,Z 548.633,A 0.000,B 0.000,C 90.000,E1 329.871} C_DIS
LIN {X -0.049,Y -512.788,Z 548.623,A 0.000,B 0.000,C 90.000,E1 328.122} C_DIS
LIN {X -0.309,Y -516.465,Z 548.611,A 0.000,B 0.000,C 90.000,E1 326.087} C_DIS
LIN {X -0.210,Y -519.121,Z 548.603,A 0.000,B 0.000,C 90.000,E1 324.609} C_DIS
LIN {X -0.109,Y -522.219,Z 548.594,A 0.000,B 0.000,C 90.000,E1 322.844} C_DIS
LIN {X -0.076,Y -526.036,Z 548.582,A 0.000,B 0.000,C 90.000,E1 320.803} C_DIS
LIN {X -0.135,Y -532.025,Z 548.566,A 0.000,B 0.000,C 90.000,E1 317.919} C_DIS
LIN {X 0.040,Y -536.621,Z 548.555,A 0.000,B 0.000,C 90.000,E1 315.891} C_DIS
LIN {X -0.062,Y -543.024,Z 548.541,A 0.000,B 0.000,C 90.000,E1 313.338} C_DIS
LIN {X -0.052,Y -545.887,Z 548.534,A 0.000,B 0.000,C 90.000,E1 312.204} C_DIS
LIN {X -0.250,Y -550.731,Z 548.524,A 0.000,B 0.000,C 90.000,E1 310.253} C_DIS
LIN {X 0.157,Y -551.403,Z 548.522,A 0.000,B 0.000,C 90.000,E1 309.930} C_DIS
LIN {X -0.300,Y -553.441,Z 548.518,A 0.000,B 0.000,C 90.000,E1 309.277} C_DIS
LIN {X 0.087,Y -554.753,Z 548.517,A 0.000,B 0.000,C 90.000,E1 308.955} C_DIS
LIN {X -0.086,Y -555.978,Z 548.515,A 0.000,B 0.000,C 90.000,E1 308.624} C_DIS
LIN {X 0.096,Y -558.197,Z 548.513,A 0.000,B 0.000,C 90.000,E1 308.257} C_DIS
LIN {X 0.071,Y -559.325,Z 548.511,A 0.000,B 0.000,C 90.000,E1 308.051} C_DIS
LIN {X -0.048,Y -561.012,Z 548.510,A 0.000,B 0.000,C 90.000,E1 307.855} C_DIS
LIN {X 0.150,Y -566.168,Z 548.507,A 0.000,B 0.000,C 90.000,E1 307.282} C_DIS
LIN {X 0.034,Y -579.629,Z 548.501,A 0.000,B 0.000,C 90.000,E1 306.171} C_DIS
LIN {X -0.234,Y -584.907,Z 548.498,A 0.000,B 0.000,C 90.000,E1 305.724} C_DIS
LIN {X -0.305,Y -591.340,Z 548.495,A 0.000,B 0.000,C 90.000,E1 305.105} C_DIS
LIN {X -0.277,Y -598.733,Z 548.491,A 0.000,B 0.000,C 90.000,E1 304.326} C_DIS
LIN {X -0.058,Y -603.569,Z 548.488,A 0.000,B 0.000,C 90.000,E1 303.785} C_DIS
LIN {X -0.183,Y -613.029,Z 548.482,A 0.000,B 0.000,C 90.000,E1 302.752} C_DIS
LIN {X 0.346,Y -620.969,Z 548.477,A 0.000,B 0.000,C 90.000,E1 301.799} C_DIS
LIN {X -0.212,Y -626.391,Z 548.473,A 0.000,B 0.000,C 90.000,E1 301.209} C_DIS
LIN {X 0.137,Y -631.220,Z 548.470,A 0.000,B 0.000,C 90.000,E1 300.541} C_DIS
LIN {X -0.039,Y -634.745,Z 548.467,A 0.000,B 0.000,C 90.000,E1 300.050} C_DIS
LIN {X 0.063,Y -638.258,Z 548.464,A 0.000,B 0.000,C 90.000,E1 299.411} C_DIS
LIN {X -0.362,Y -641.197,Z 548.460,A 0.000,B 0.000,C 90.000,E1 298.821} C_DIS
LIN {X 0.282,Y -645.611,Z 548.453,A 0.000,B 0.000,C 90.000,E1 297.513} C_DIS
LIN {X -0.051,Y -648.180,Z 548.449,A 0.000,B 0.000,C 90.000,E1 296.796} C_DIS
LIN {X 0.124,Y -649.313,Z 548.446,A 0.000,B 0.000,C 90.000,E1 296.283} C_DIS
